// TwinCAT 3 PLC project MC2
// Title: Tc_MC2
// Company: NewEngineer
// Author: Tc_MC2
// ProjectVersion: 0.1.1.1
// Description: https://github.com/phucpha
// ProgramVersion: 3.1.4024.0
// libraries:
//   Tc2_MC2, * (Beckhoff Automation GmbH)
//   Tc2_Standard, * (Beckhoff Automation GmbH)
//   Tc2_System, * (Beckhoff Automation GmbH)
//   Tc3_EventLogger, * (Beckhoff Automation GmbH)
//   Tc3_Mc3Definitions, * (Beckhoff Automation GmbH)
//   Tc3_Module, * (Beckhoff Automation GmbH)
//   Tc_Utilities, * (NewEngineer)
// project tree:
//   DUTs/CAextension/ E_AxisStateCA.TcDUT
//   DUTs/CA/ E_AxesGroupCAMethodState.TcDUT, E_AxesGroupCAState.TcDUT, E_AxesGroupCAStateAborting.TcDUT, E_AxesGroupCAStateInit.TcDUT, E_AxesGroupCAStatePlcOpen.TcDUT
//   DUTs/Universal Axis/ E_AxisJogDirection.TcDUT, E_AxisState.TcDUT, E_AxisStateInit.TcDUT, E_AxisStatePlcOpen.TcDUT
//   DUTs/Visu/ E_VisuCtrlAxisImgType.TcDUT (not stored), E_VisuCtrlAxisJogMode.TcDUT (not stored), E_VisuCtrlSingleAxisState.TcDUT (not stored), ST_VisuCtrlAxisFrame.TcDUT (not stored)
//   POUs/AxesGroup/ FB_AxesGroupCA.TcPOU, I_AxesGroupCA.TcIO
//   POUs/Axis/ FB_AxisServo.TcPOU, FB_AxisServoCA.TcPOU, FB_UniversalAxis.TcPOU, I_UniversalAxis.TcIO, I_UniversalAxisCA.TcIO
//   Version/ Global_Version.TcGVL
// real-time tasks:
//   TASK PlcTask: cycle T#10ms, priority 20, ADS port 350

// ---- DUTs/CAextension/E_AxisStateCA.TcDUT
{attribute 'strict'}
TYPE E_AxisStateCA :
(
	AXIS_CA_IDLE				:= 0,
	AXIS_CA_MOVE_ABSOLUTE 		:= 10,
	AXIS_CA_MOVE_ABSOLUTE_DONE 	:= 20,
	AXIS_CA_MOVE_RELATIVE 		:= 30,
	AXIS_CA_MOVE_RELATIVE_DONE 	:= 40,
	AXIS_CA_HALT				:= 50,
	AXIS_CA_HALT_DONE			:= 60
);
END_TYPE

// ---- DUTs/CA/E_AxesGroupCAMethodState.TcDUT
{attribute 'strict'}
TYPE E_AxesGroupCAMethodState :
(
	AXES_GROUP_METHOD_EXECUTE 	:= 0,	(* Reseting all fubs *)
	AXES_GROUP_METHOD_DONE		:= 10	(* Enabling axes group *)
);
END_TYPE

// ---- DUTs/CA/E_AxesGroupCAState.TcDUT
{attribute 'strict'}
TYPE E_AxesGroupCAState :
(
	AXES_GROUP_UNINITIALIZED 		:= 0,	(* Axes group is disabled, not ready to work *)
	AXES_GROUP_INITIALIZING 		:= 10,	(* Axes group is preprating to work *)
	AXES_GROUP_READY_INITIALIZED	:= 20,	(*  *)
	AXES_GROUP_IDLE 				:= 30,	(* Axes group ready to work, enabled *)
	AXES_GROUP_ADD					:= 40,	(* Adding axis to axes group *)
	AXES_GROUP_ADD_DONE				:= 50,	(* Adding axis to axes group done *)
	AXES_GROUP_REMOVE				:= 60,	(* Removeing axis from axes group *)
	AXES_GROUP_REMOVE_DONE			:= 70,	(* Removing axis from axes group done *)
	AXES_GROUP_REMOVE_ALL			:= 80,	(* Remoing all axis from axes group *)
	AXES_GROUP_REMOVE_ALL_DONE		:= 90,	(* Removing all axis from axes group done *)
	AXES_GROUP_ENABLE				:= 100,	(* Enabling axes group *)
	AXES_GROUP_ENABLE_DONE			:= 110,	(* Enabling axes group done *)
	AXES_GROUP_DISABLE				:= 120,	(* Disabling axes group *)
	AXES_GROUP_DISABLE_DONE			:= 130,	(* Disabling axes group done *)
	AXES_GROUP_RESET				:= 140,	(* Reseting funcion block *)
	AXES_GROUP_RESET_DONE			:= 150,	(* Reseting function block done *)
	AXES_GROUP_HALT					:= 160,	(* Halt axes group *)
	AXES_GROUP_HALT_DONE			:= 170,	(* Halt axes group done *)
	AXES_GROUP_STOP					:= 180,	(* Stop axes group *)
	AXES_GROUP_STOP_DONE			:= 190,	(* Stop axes group done *)
	AXES_GROUP_UNLOCK				:= 200,	(* Unlock axes group after stop *)
	AXES_GROUP_UNLOCK_DONE			:= 210,	(* Unlock axes group after stop done *)
	AXES_GROUP_ABORTING				:= -10	(* Aborting *)
);
END_TYPE

// ---- DUTs/CA/E_AxesGroupCAStateAborting.TcDUT
{attribute 'strict'}
TYPE E_AxesGroupCAStateAborting :
(
	AXES_GROUP_ABORTING_RESET_FBS 		:= 0,	(* Reseting all function blocks used inside function block *)
	AXES_GROUP_ABORTING_REMOVE_ALL		:= 10,	(* Removing all axis from axes group  *)
	AXES_GROUP_ABORTING_RESET_ERRORS	:= 20,	(* Reseting axes group errors *)
	AXES_GROUP_ABORTING_DISABLE			:= 30,	(* Disabling axes group *)
	AXES_GROUP_ABORTING_DONE			:= 40	(* Aborting procedure finished *)
);
END_TYPE

// ---- DUTs/CA/E_AxesGroupCAStateInit.TcDUT
{attribute 'strict'}
TYPE E_AxesGroupCAStateInit :
(
	AXES_GROUP_INIT_RESET 	:= 0,	(* Reseting all fubs *)
	AXES_GROUP_INIT_ENABLE	:= 10,	(* Enabling axes group *)
	AXES_GROUP_INIT_DONE	:= 20	(* Initialization procedure done*)
);
END_TYPE

// ---- DUTs/CA/E_AxesGroupCAStatePlcOpen.TcDUT
{attribute 'strict'}
TYPE E_AxesGroupCAStatePlcOpen :
(
	PLCOPEN_AXES_GROUP_DISABLED 	:= 0,	(* Axes group is disabled *)
	PLCOPEN_AXES_GROUP_NOT_READY 	:= 10,	(* Axes group is not ready to work*)
	PLCOPEN_AXES_GROUP_STANDBY 		:= 20,	(* Axes group is enabled and waiting for commands*)
	PLCOPEN_AXES_GROUP_MOVING 		:= 30,	(* Axes group is moving *)
	PLCOPEN_AXES_GROUP_STOPPING 	:= 40,	(* Axes group is stopping *)
	PLCOPEN_AXES_GROUP_ERROR		:= 50	(* Axes group is in error state*)
);
END_TYPE

// ---- DUTs/Universal Axis/E_AxisJogDirection.TcDUT
{attribute 'strict'}
TYPE E_AxisJogDirection :
(
	AXIS_JOG_DIR_POSITIVE := 0,	(* Perform jog in positive direction *)
	AXIS_JOG_DIR_NEGATIVE := 10	(* Perform jog in negative direction *)
);
END_TYPE

// ---- DUTs/Universal Axis/E_AxisState.TcDUT
{attribute 'strict'}
TYPE E_AxisState :
(
	AXIS_UNINITIALIZED		:= 0,	(* Axis is not prepared to work - power is off *)
	AXIS_INITIALIZING		:= 10,	(* Axis is preparing to power - reset FB and power on *)
	AXIS_READY_INITIALIZED	:= 20,	(*  *)
	AXIS_IDLE				:= 30,	(* Axis is ready for orders *)
	AXIS_HOME				:= 40,	(* Axis is homing to reference point *)
	AXIS_HOME_DONE			:= 50,	(* Axis homing procedure has finished - fererence position has been found *)
	AXIS_MOVE_VELOCITY		:= 60,	(* Axis started continous motion to setpoint velocity - accelerating *)
	AXIS_MOVE_VELOCITY_DONE	:= 70,	(* Axis reached constant setpoint velocity for continous motion *)
	AXIS_MOVE_ABSOLUTE		:= 80,	(* Axis is moving to absolute position - discrete motion *)
	AXIS_MOVE_ABSOLUTE_DONE	:= 90,	(* Axis movement to absolute position finished *)
	AXIS_MOVE_ADDITIVE		:= 100,	(* Axis relative movement by desired distance *)
	AXIS_MOVE_ADDITIVE_DONE	:= 110,	(* Axis relative relative movement by desired distance finished *)
	AXIS_MOVE_RELATIVE		:= 120,	(* Axis relative movement by desired distance *)
	AXIS_MOVE_RELATIVE_DONE	:= 130,	(* Axis relative relative movement by desired distance finished *)
	AXIS_MOVE_JOG			:= 140,	(* Axis manual move using jog function *)
	AXIS_MOVE_JOG_DONE		:= 150,	(* Axis jog done *)
	AXIS_STOP				:= 160,	(* Axis is stopping *)
	AXIS_STOP_DONE			:= 170,	(* Axis stopped *)
	AXIS_HALT				:= 180,	(* Axis halts started motion command *)
	AXIS_HALT_DONE			:= 190,	(* Axis motion halted *)
	AXIS_RESET				:= 200,	(* Axis is resseting all function blocks and occured errors *)
	AXIS_RESET_DONE			:= 210,	(* Axis reset procedure done *)
	AXIS_COUPLE				:= 220, (* Axis is synchronizing to another master axis *)
	AXIS_COUPLE_DONE		:= 230,	(* Axis coupled to another master axis*)
	AXIS_DECOUPLE			:= 240,	(* Axis is decoupling from synchronized motion *)
	AXIS_DECOUPLE_DONE		:= 250,	(* Axis decoupled from synchronizing motion*)
	AXIS_UNLOCK				:= 260,	(* Axis is unlocking after stop command *)
	AXIS_UNLOCK_DONE		:= 270,	(* Axis unlocked after stop command *)
	AXIS_EXTENSION			:= 999,	(* Special state used by child FB's to implement additional states *)
	AXIS_ABORTING			:= -10	(* Aborting *)
);
END_TYPE

// ---- DUTs/Universal Axis/E_AxisStateInit.TcDUT
{attribute 'strict'}
TYPE E_AxisStateInit :
(
	AXIS_INIT_RESET		:= 0,	(* Reseting all function blocks *)
	AXIS_INIT_POWER_ON	:= 10,	(* Powering on the axis *)
	AXIS_INIT_DONE		:= 20	(* Initialization done *)
);
END_TYPE

// ---- DUTs/Universal Axis/E_AxisStatePlcOpen.TcDUT
{attribute 'strict'}
TYPE E_AxisStatePlcOpen :
(
	AXIS_PLCOPEN_DISABLED				:= 0,	(* Axis power controler if of *)
	AXIS_PLCOPEN_STANDSTILL				:= 10,	(* Axis is powered on *)
	AXIS_PLCOPEN_HOMING					:= 20,	(* Axis performs homing procedure *)
	AXIS_PLCOPEN_STOPPING				:= 30,	(* Axis is stopping the movement *)
	AXIS_PLCOPEN_CONTINUOUS_MOTION		:= 40,	(* Axis is moving continuosly with constant speed *)
	AXIS_PLCOPEN_DISCRETE_MOTION		:= 50,	(* Axis is moving from point to point *)
	AXIS_PLCOPEN_SYNCHRONIZED_MOTION 	:= 60,	(* Axis is moving in synchronized motion to master *)
	AXIS_PLCOPEN_ERRORSTOP				:= 70	(* Axis stoped because of error *)
);
END_TYPE

// ---- Version/Global_Version.TcGVL
{attribute 'TcGenerated'}
{attribute 'no-analysis'}
{attribute 'linkalways'}
// This function has been automatically generated from the project information.
VAR_GLOBAL CONSTANT
	{attribute 'const_non_replaced'}
	stLibVersion_Tc_MC2 : ST_LibVersion := (iMajor := 0, iMinor := 1, iBuild := 1, iRevision := 1, nFlags := 0, sVersion := '0.1.1.1');
END_VAR

// ---- POUs/AxesGroup/I_AxesGroupCA.TcIO
INTERFACE I_AxesGroupCA

PROPERTY Active : REFERENCE TO BOOL
GET
END_GET
END_PROPERTY

PROPERTY AxesGroupRef : REFERENCE TO AXES_GROUP_REF
GET
END_GET
END_PROPERTY

PROPERTY AxesInGroup : REFERENCE TO UINT
GET
END_GET
END_PROPERTY

PROPERTY AxisAdded : REFERENCE TO BOOL
GET
END_GET
END_PROPERTY

PROPERTY AxisRemoved : REFERENCE TO BOOL
GET
END_GET
END_PROPERTY

PROPERTY Busy : REFERENCE TO BOOL
GET
END_GET
END_PROPERTY

PROPERTY Deceleration : LREAL
GET
END_GET
SET
END_SET
END_PROPERTY

PROPERTY Error : REFERENCE TO BOOL
GET
END_GET
END_PROPERTY

PROPERTY ErrorID : REFERENCE TO UDINT
GET
END_GET
END_PROPERTY

PROPERTY GroupEnabled : REFERENCE TO BOOL
GET
END_GET
END_PROPERTY

PROPERTY GroupLocked : REFERENCE TO BOOL
GET
END_GET
END_PROPERTY

PROPERTY Jerk : LREAL
GET
END_GET
SET
END_SET
END_PROPERTY

METHOD MR_Abort : BOOL
VAR_INPUT
END_VAR
END_METHOD

METHOD MR_Add : BOOL
VAR_INPUT
	stInternalAxisRef	: AXIS_REF;
	iAxisIdentyficator	: UINT;
END_VAR
END_METHOD

METHOD MR_Disable : BOOL
VAR_INPUT
END_VAR
END_METHOD

METHOD MR_Enable : BOOL
VAR_INPUT
END_VAR
END_METHOD

METHOD MR_FirstCycle
VAR_INPUT
	sName 			: STRING;	(* Default axes group object name *)
	lrDeceleration 	: LREAL;	(* Default axes group object deceleration *)
	lrJerk			: LREAL;	(* Default axes group object jerk *)
END_VAR
END_METHOD

METHOD MR_Halt : BOOL
VAR_INPUT
END_VAR
END_METHOD

METHOD MR_Init : BOOL
VAR_INPUT
END_VAR
END_METHOD

METHOD MR_Remove : BOOL
VAR_INPUT
	iAxisIdentyficator	: UINT;
END_VAR
END_METHOD

METHOD MR_RemoveAll : BOOL
VAR_INPUT
END_VAR
END_METHOD

METHOD MR_Reset : BOOL
VAR_INPUT
END_VAR
END_METHOD

METHOD MR_Stop : BOOL
VAR_INPUT
END_VAR
END_METHOD

METHOD MR_Unlock : BOOL
VAR_INPUT
END_VAR
END_METHOD

PROPERTY Name : STRING
GET
END_GET
SET
END_SET
END_PROPERTY

PROPERTY RemovedAll : REFERENCE TO BOOL
GET
END_GET
END_PROPERTY

PROPERTY State : REFERENCE TO E_AxesGroupCAState
GET
END_GET
END_PROPERTY

PROPERTY StatePlcOpen : REFERENCE TO E_AxesGroupCAStatePlcOpen
GET
END_GET
END_PROPERTY

END_INTERFACE

// ---- POUs/Axis/I_UniversalAxis.TcIO
INTERFACE I_UniversalAxis

PROPERTY Acceleration : LREAL
GET
END_GET
SET
END_SET
END_PROPERTY

PROPERTY Active : REFERENCE TO BOOL
GET
END_GET
END_PROPERTY

PROPERTY ActualPosition : REFERENCE TO LREAL
GET
END_GET
END_PROPERTY

PROPERTY ActualVelocity : REFERENCE TO LREAL
GET
END_GET
END_PROPERTY

PROPERTY AxisErrorID : REFERENCE TO UDINT
GET
END_GET
END_PROPERTY

PROPERTY AxisRef : AXIS_REF
GET
END_GET
SET
END_SET
END_PROPERTY

PROPERTY BufferMode : MC_BufferMode
GET
END_GET
SET
END_SET
END_PROPERTY

PROPERTY Busy : REFERENCE TO BOOL
GET
END_GET
END_PROPERTY

PROPERTY Deceleration : LREAL
GET
END_GET
SET
END_SET
END_PROPERTY

PROPERTY Direction : Tc2_MC2.MC_Direction
GET
END_GET
SET
END_SET
END_PROPERTY

PROPERTY Error : REFERENCE TO BOOL
GET
END_GET
END_PROPERTY

PROPERTY ErrorID : REFERENCE TO UDINT
GET
END_GET
END_PROPERTY

PROPERTY Halted : REFERENCE TO BOOL
GET
END_GET
END_PROPERTY

PROPERTY InPosition : REFERENCE TO BOOL
GET
END_GET
END_PROPERTY

PROPERTY InVelocity : REFERENCE TO BOOL
GET
END_GET
END_PROPERTY

PROPERTY IsHomed : REFERENCE TO BOOL
GET
END_GET
END_PROPERTY

PROPERTY Jerk : LREAL
GET
END_GET
SET
END_SET
END_PROPERTY

PROPERTY JogAcceleration : LREAL
GET
END_GET
SET
END_SET
END_PROPERTY

PROPERTY JogDeceleration : LREAL
GET
END_GET
SET
END_SET
END_PROPERTY

PROPERTY JogDirection : E_AxisJogDirection
GET
END_GET
SET
END_SET
END_PROPERTY

PROPERTY JogDone : REFERENCE TO BOOL
GET
END_GET
END_PROPERTY

PROPERTY JogJerk : LREAL
GET
END_GET
SET
END_SET
END_PROPERTY

PROPERTY JogMode : E_JogMode
GET
END_GET
SET
END_SET
END_PROPERTY

PROPERTY JogPosition : LREAL
GET
END_GET
SET
END_SET
END_PROPERTY

PROPERTY JogVelocity : LREAL
GET
END_GET
SET
END_SET
END_PROPERTY

PROPERTY LagError : LREAL
GET
END_GET
END_PROPERTY

PROPERTY MoveActive : REFERENCE TO BOOL
GET
END_GET
END_PROPERTY

METHOD MR_Abort : BOOL
END_METHOD

METHOD MR_FirstCycle
VAR_INPUT
	sName 				: STRING; 	(* Axis object name *)
	sMeasurementUnits	: STRING;	(* Measurement units used by axis *)
	bModulo				: BOOL;		(* Axis is periodic *)
END_VAR
END_METHOD

METHOD MR_Halt : BOOL
END_METHOD

METHOD MR_Home : BOOL
VAR_INPUT
	lrHomePosition : LREAL;
END_VAR
END_METHOD

METHOD MR_Init : BOOL
END_METHOD

METHOD MR_Jog : BOOL
VAR_INPUT
	//lrJogPosition : LREAL;
	//eJogDirection : E_AxisJogDirection;
	//eJogMode	  : E_JogMode;
	bJogActive	  : BOOL;
END_VAR
END_METHOD

METHOD MR_MoveAbsolute : BOOL
VAR_INPUT
	lrAbsolutePosition : LREAL;
END_VAR
END_METHOD

METHOD MR_MoveAdditive : BOOL
VAR_INPUT
	lrRelativeDistance : LREAL;
END_VAR
END_METHOD

METHOD MR_MoveRelative : BOOL
VAR_INPUT
	lrRelativeDistance : LREAL;
END_VAR
END_METHOD

METHOD MR_MoveVelocity : BOOL
END_METHOD

METHOD MR_Reset : BOOL
END_METHOD

METHOD MR_Stop : BOOL
END_METHOD

PROPERTY Name : STRING
GET
END_GET
SET
END_SET
END_PROPERTY

PROPERTY Options : ST_MoveOptions
GET
END_GET
SET
END_SET
END_PROPERTY

PROPERTY Override : LREAL
GET
END_GET
SET
END_SET
END_PROPERTY

PROPERTY PowerOn : REFERENCE TO BOOL
GET
END_GET
END_PROPERTY

PROPERTY SetpointPosition : LREAL
GET
END_GET
END_PROPERTY

PROPERTY SetpointVelocity : LREAL
GET
END_GET
END_PROPERTY

PROPERTY State : REFERENCE TO E_AxisState
GET
END_GET
END_PROPERTY

PROPERTY StatePlcOpen : REFERENCE TO E_AxisStatePlcOpen
GET
END_GET
END_PROPERTY

PROPERTY StopDeceleration : LREAL
GET
END_GET
SET
END_SET
END_PROPERTY

PROPERTY StopJerk : LREAL
GET
END_GET
SET
END_SET
END_PROPERTY

PROPERTY Stopped : REFERENCE TO BOOL
GET
END_GET
END_PROPERTY

PROPERTY Unit : STRING
GET
END_GET
SET
END_SET
END_PROPERTY

PROPERTY Velocity : LREAL
GET
END_GET
SET
END_SET
END_PROPERTY

END_INTERFACE

// ---- POUs/Axis/I_UniversalAxisCA.TcIO
INTERFACE I_UniversalAxisCA EXTENDS I_UniversalAxis

PROPERTY DirectionCA : Tc3_Mc3Definitions.MC_DIRECTION
GET
END_GET
SET
END_SET
END_PROPERTY

PROPERTY Gap : MC_LREAL
GET
END_GET
SET
END_SET
END_PROPERTY

PROPERTY HaltedCA : REFERENCE TO BOOL
GET
END_GET
END_PROPERTY

METHOD MR_HaltCA : BOOL
VAR_INPUT
END_VAR
END_METHOD

METHOD MR_MoveAbsoluteCA : BOOL
VAR_INPUT
	lrAbsolutePosition : LREAL;
END_VAR
END_METHOD

METHOD MR_MoveRelativeCA : BOOL
VAR_INPUT
	lrRelativeDistance : LREAL;
END_VAR
END_METHOD

PROPERTY StateCA : REFERENCE TO E_AxisStateCA
GET
END_GET
END_PROPERTY

END_INTERFACE

// ---- POUs/AxesGroup/FB_AxesGroupCA.TcPOU
(*
:Description: This function block is used to control collision avoidance axes group.
*)
FUNCTION_BLOCK FB_AxesGroupCA IMPLEMENTS I_AxesGroupCA
VAR
	bFirstCycle				: BOOL := TRUE;						(* First cycle bit *)	
	sName 					: STRING;							(* Axes group name for other utilities *)
	
	(* Hardware links *)
	stAxesGroupRef 			: AXES_GROUP_REF;					(* Axes group reference object *)
	stInternalAxisRef 		: AXIS_REF;							(* Internal axis reference object *)
	
	(* Internal commands *)
	bInit 					: BOOL;								(* Power on axis and prepare to work *)
	bAbort 					: BOOL;								(* Power off axis and reset status flags *)
	bReset 					: BOOL;								(* Reset axis and return to READY state *)
	bAdd 					: BOOL;								(* Add axis to the group *)
	bRemove 				: BOOL;								(* Remove axis from the group *)
	bRemoveAll 				: BOOL;								(* Remove all axes from the group *)
	bEnable 				: BOOL;								(* Enable the group *)
	bDisable 				: BOOL;								(* Disable the group *)
	bGroupHalt				: BOOL;								(* Halt all axes in group *)
	bGroupStop				: BOOL;								(* Stop all axes in group *)
	bGroupUnlock			: BOOL;								(* Unlock axes group after stop *)
	
	(* Internal parameters *)
	iIdentInGroup			: UDINT;							(* An axis identyficator *)
	lrDeceleration			: LREAL;							(* Decelearion of all axes in group *)
	lrJerk					: LREAL;							(* Jerk of all axes in group *)
	
	(* Internal status *)
	bActive					: BOOL;
	bBusy					: BOOL;								(* Function block currently executes one of the requests *)
	bError 					: BOOL;								(* Error status flag *)
	iErrorID 				: UDINT;							(* Error ID *)
	bResetDone				: BOOL;								(* All internal errors of a group and all axes belonging to the group reset *)	
	bAxisAdded				: BOOL;								(* Axis added to the group *)
	bAxisRemoved			: BOOL;								(* Axis removed from the group *)
	bRemovedAll				: BOOL;								(* Removing all axes and disabling the group *)
	bGroupEnabled			: BOOL;								(* Axes group enabled *)
	bGroupHalted			: BOOL;								(* Axes group halted *)
	bGroupStopped			: BOOL;								(* Axes group stopped *)
	iAxesInGroup			: UINT;								(* Amount of the axes in the group *)
	bGroupLocked			: BOOL;								(* Group locked by stop function *)
	eStatePlcOpen 			: E_AxesGroupCAStatePlcOpen;
	eAxesGroupState 		: E_AxesGroupCAState;
	eAxesGroupStateInit		: E_AxesGroupCAStateInit;
	eAxesGroupStateAbort	: E_AxesGroupCAStateAborting;
	eAxesGroupMethodState	: E_AxesGroupCAMethodState;
	
	
	(* Function blocks *)
	fbMcAddAxisToGroup		: MC_AddAxisToGroup;				(* FB to add an axis to the group *)
	fbMcRemoveAxisFromGroup	: MC_RemoveAxisFromGroup;			(* FB to remove an axis from the group *)
	fbMcUngroupAllAxes 		: MC_UngroupAllAxes;				(* FB to ungroup all axes from the group *)
	
	fbMcGroupEnable 		: MC_GroupEnable;					(* FB to enable the group *)
	fbMcGroupDisable 		: MC_GroupDisable;					(* FB to disable the group *)
	
	fbMcGroupReadStatus		: MC_GroupReadStatus;				(* FB to read current axes group status *)
	fbMcGroupReadError		: MC_GroupReadError;				(* FB to read axes group error *)
	fbMcGroupReset 			: MC_GroupReset;					(* FB to reset axes group *)
	
	fbMcGroupHalt			: MC_GroupHalt;						(* FB to halt all axes in group *)
	fbMcGroupStop			: MC_GroupStop;						(* FB to stop all axes in group *)
	
	(* Tc3 EventLogger - messages *)
	fbAlarmGroupReset		: FB_TcAlarm;						(*  *)
	fbAlarmUngroupAll		: FB_TcAlarm;						(*  *)
	fbAlarmGroupDisable		: FB_TcAlarm;						(*  *)
	fbAlarmAddAxisToGroup	: FB_TcAlarm;						(*  *)
	fbAlarmGroupEnable		: FB_TcAlarm;						(*  *)
	fbAlarmRemoveFromGroup	: FB_TcAlarm;						(*  *)
	
	bResetConfirmation 		: BOOL;
	bGroupHaltLog			: BOOL;
	bGroupStopLog			: BOOL;
	
	rtError					: R_TRIG; 				(* Rising edge trigger for function block error *)
	
END_VAR

(* Run first cycle procedure *)
IF bFirstCycle THEN
	bFirstCycle := FALSE;
		
	fbAlarmGroupReset.CreateEx( stEventEntry := TC_EVENTS.ShellAxesGroupEventClass.GroupReset, 
									bWithConfirmation := 1,
									ipSourceInfo := 0);
									
	fbAlarmUngroupAll.CreateEx( stEventEntry := TC_EVENTS.ShellAxesGroupEventClass.UngroupAll, 
									bWithConfirmation := 1,
									ipSourceInfo := 0);
		
	fbAlarmGroupDisable.CreateEx( stEventEntry := TC_EVENTS.ShellAxesGroupEventClass.GroupDisable, 
									bWithConfirmation := 1,
									ipSourceInfo := 0);
									
	fbAlarmAddAxisToGroup.CreateEx( stEventEntry := TC_EVENTS.ShellAxesGroupEventClass.AddAxisToGroup, 
									bWithConfirmation := 1,
									ipSourceInfo := 0);
		
	fbAlarmGroupEnable.CreateEx( stEventEntry := TC_EVENTS.ShellAxesGroupEventClass.GroupEnable, 
									bWithConfirmation := 1,
									ipSourceInfo := 0);
									
	fbAlarmRemoveFromGroup.CreateEx( stEventEntry := TC_EVENTS.ShellAxesGroupEventClass.RemoveFromGroup, 
									bWithConfirmation := 1,
									ipSourceInfo := 0);
									
END_IF

(* Reading the group status from group reference *)
fbMcGroupReadStatus( AxesGroup := stAxesGroupRef, Enable := TRUE);

(* Setting the PLCOpen group status*)
IF fbMcGroupReadStatus.Valid THEN
	IF fbMcGroupReadStatus.GroupDisabled THEN
		eStatePlcOpen := PLCOPEN_AXES_GROUP_DISABLED;
		
	ELSIF fbMcGroupReadStatus.GroupErrorStop THEN
		eStatePlcOpen := PLCOPEN_AXES_GROUP_ERROR;
		
	ELSIF fbMcGroupReadStatus.GroupStandby THEN
		eStatePlcOpen := PLCOPEN_AXES_GROUP_STANDBY;
		
	ELSIF fbMcGroupReadStatus.GroupMoving THEN
		eStatePlcOpen := PLCOPEN_AXES_GROUP_MOVING;
		
	ELSIF fbMcGroupReadStatus.GroupStopping THEN
		eStatePlcOpen := PLCOPEN_AXES_GROUP_STOPPING;
		
	END_IF
END_IF

(* Reading errors *)
fbMcGroupReadError( AxesGroup := stAxesGroupRef, Enable := TRUE);

IF fbMcGroupReadError.Valid THEN
	iErrorID := fbMcGroupReadError.GroupErrorId;
END_IF


(* Report errors that occur *)
rtError(CLK:=bError);

IF rtError.Q THEN 
	fbMachineLogger.MR_AddLogs(FUN_MergeStrings5(sName, ' : Error occured (error ID: ', UDINT_TO_STRING(iErrorID), ')', ''));

END_IF

(* Execute state machine *)
StateMachine();

PROPERTY Active : REFERENCE TO BOOL
GET
Active REF= bActive;
END_GET
END_PROPERTY

PROPERTY AxesGroupRef : REFERENCE TO Tc3_McCoordinatedMotion.AXES_GROUP_REF
GET
AxesGroupRef REF= stAxesGroupRef;
END_GET
END_PROPERTY

PROPERTY AxesInGroup : REFERENCE TO UINT
GET
AxesInGroup REF= iAxesInGroup;
END_GET
END_PROPERTY

PROPERTY AxisAdded : REFERENCE TO BOOL
GET
AxisAdded REF= bAxisAdded;
END_GET
END_PROPERTY

PROPERTY AxisRemoved : REFERENCE TO BOOL
GET
AxisRemoved REF= bAxisRemoved;
END_GET
END_PROPERTY

PROPERTY Busy : REFERENCE TO BOOL
GET
Busy REF= bBusy;
END_GET
END_PROPERTY

(* Decelearion of all axes in group *)
PROPERTY Deceleration : LREAL
GET
Deceleration := lrDeceleration;
END_GET
SET
lrDeceleration := Deceleration;
END_SET
END_PROPERTY

PROPERTY Error : REFERENCE TO BOOL
GET
Error REF= bError;
END_GET
END_PROPERTY

PROPERTY ErrorID : REFERENCE TO UDINT
GET
ErrorID REF= iErrorID;
END_GET
END_PROPERTY

PROPERTY GroupEnabled : REFERENCE TO BOOL
GET
GroupEnabled REF= bGroupEnabled;
END_GET
END_PROPERTY

PROPERTY GroupHalted : REFERENCE TO BOOL
GET
GroupHalted REF= bGroupHalted;
END_GET
END_PROPERTY

PROPERTY GroupLocked : REFERENCE TO BOOL
GET
GroupLocked REF= bGroupLocked;
END_GET
END_PROPERTY

PROPERTY GroupStopped : REFERENCE TO BOOL
GET
GroupStopped REF= bGroupStopped;
END_GET
END_PROPERTY

(* Jerk of all axes in group *)
PROPERTY Jerk : LREAL
GET
Jerk := lrJerk;
END_GET
SET
lrJerk := Jerk;
END_SET
END_PROPERTY

METHOD MR_Abort : BOOL
IF eAxesGroupState >= AXES_GROUP_IDLE THEN
	bBusy := TRUE;
	bAbort := TRUE;
	eAxesGroupStateAbort := AXES_GROUP_ABORTING_RESET_FBS;
	eAxesGroupState := AXES_GROUP_ABORTING;	
	
	fbMachineLogger.MR_AddLogs(CONCAT(sName,' : abort requested'));			

ELSIF eAxesGroupState = AXES_GROUP_ABORTING AND eAxesGroupStateAbort = AXES_GROUP_ABORTING_DONE THEN
	bActive := FALSE;
	bAbort := FALSE;	
	MR_Abort := TRUE;
	bBusy := FALSE;
	
	fbMachineLogger.MR_AddLogs(CONCAT(sName,' : abort done'));	

END_IF
END_METHOD

METHOD MR_Add : BOOL
VAR_INPUT
	stInternalAxisRef	: AXIS_REF;
	iAxisIdentyficator	: UINT;
END_VAR
IF eAxesGroupState = AXES_GROUP_IDLE THEN
	bBusy 			:= TRUE;
	bAdd 			:= TRUE;
	
	bAxisAdded 		:= FALSE;
	bAxisRemoved 	:= FALSE;
	bRemovedAll 	:= FALSE;
	bResetDone		:= FALSE;
	
	THIS^.stInternalAxisRef := stInternalAxisRef;
	iIdentInGroup := iAxisIdentyficator;
	
	eAxesGroupState := AXES_GROUP_ADD;
	fbMachineLogger.MR_AddLogs(CONCAT(sName,' : axes group addition requested'));			
	
ELSIF eAxesGroupState = AXES_GROUP_ADD_DONE THEN
	bAdd 			:= FALSE;
	
	MR_Add 			:= TRUE;
	bAxisAdded 		:= TRUE;
	iAxesInGroup 	:= iAxesInGroup + 1;

	bBusy			:= FALSE;

	fbMachineLogger.MR_AddLogs(CONCAT(sName,' : axes group addition done'));			
	
END_IF
END_METHOD

METHOD MR_Disable : BOOL
VAR_INPUT
END_VAR
IF eAxesGroupState = AXES_GROUP_IDLE THEN
	bBusy 			:= TRUE;
	bDisable 		:= TRUE;
	
	bAxisAdded 		:= FALSE;
	bAxisRemoved 	:= FALSE;
	bRemovedAll 	:= FALSE;
	bResetDone		:= FALSE;
	
	eAxesGroupState := AXES_GROUP_DISABLE;
	fbMachineLogger.MR_AddLogs(CONCAT(sName,' : axes group disablement requested'));				
	
ELSIF eAxesGroupState = AXES_GROUP_DISABLE_DONE THEN
	bDisable 		:= FALSE;
	
	MR_Disable 		:= TRUE;
	bGroupEnabled	:= FALSE;
	
	bBusy 			:= FALSE;
	
	fbMachineLogger.MR_AddLogs(CONCAT(sName,' : axes group disablement done'));			
	
END_IF
END_METHOD

METHOD MR_Enable : BOOL
VAR_INPUT
END_VAR
IF eAxesGroupState = AXES_GROUP_IDLE THEN
	bBusy			:= TRUE;
	bEnable 		:= TRUE;
	
	bAxisAdded 		:= FALSE;
	bAxisRemoved 	:= FALSE;
	bRemovedAll 	:= FALSE;
	bResetDone		:= FALSE;
	
	eAxesGroupState := AXES_GROUP_ENABLE;
	fbMachineLogger.MR_AddLogs(CONCAT(sName,' : axes group enablement requested'));
	
ELSIF eAxesGroupState = AXES_GROUP_ENABLE_DONE THEN
	bEnable 		:= FALSE;
	MR_Enable 		:= TRUE;
	bGroupEnabled 	:= TRUE;
	bBusy 			:= FALSE;
	fbMachineLogger.MR_AddLogs(CONCAT(sName,' : axes group enablement done'));
	
END_IF
END_METHOD

METHOD MR_FirstCycle
VAR_INPUT
	sName 			: STRING;	(* Default axes group object name *)
	lrDeceleration 	: LREAL;	(* Default axes group object deceleration *)
	lrJerk			: LREAL;	(* Default axes group object jerk *)
END_VAR
THIS^.sName := sName;
THIS^.lrDeceleration := lrDeceleration;
THIS^.lrJerk := lrJerk;
END_METHOD

METHOD MR_Halt : BOOL
VAR_INPUT
END_VAR
IF eAxesGroupState >= AXES_GROUP_IDLE AND eAxesGroupState <> AXES_GROUP_HALT_DONE THEN
	bBusy := TRUE;
	
	IF NOT bGroupHaltLog THEN 
		fbMachineLogger.MR_AddLogs(CONCAT(sName,' : halt requested'));
		bGroupHaltLog := TRUE;
	END_IF
	
	bGroupHalt := TRUE;
	MR_Halt := FALSE;
	eAxesGroupState := AXES_GROUP_HALT;
	
ELSIF eAxesGroupState = AXES_GROUP_HALT_DONE THEN
	bGroupHalt := FALSE;
	MR_Halt := TRUE;
	bGroupHaltLog := FALSE;
	bBusy := FALSE;
	
	fbMachineLogger.MR_AddLogs(CONCAT(sName,' : halt done'));
	
END_IF
END_METHOD

METHOD MR_Init : BOOL
IF eAxesGroupState = AXES_GROUP_UNINITIALIZED THEN
	bBusy := TRUE;
	bActive := TRUE;
	bInit := TRUE;
	MR_Init := FALSE;
	eAxesGroupState := AXES_GROUP_INITIALIZING;
	fbMachineLogger.MR_AddLogs(CONCAT(sName,' : initialization requested'));
	
ELSIF eAxesGroupState = AXES_GROUP_INITIALIZING AND eAxesGroupStateInit = AXES_GROUP_INIT_DONE THEN
	bInit := FALSE;
	MR_Init := TRUE;
	bBusy := FALSE;

	fbMachineLogger.MR_AddLogs(CONCAT(sName,' : initialization done'));	

END_IF
END_METHOD

METHOD MR_Remove : BOOL
VAR_INPUT
	iAxisIdentyficator	: UINT;
END_VAR
IF eAxesGroupState = AXES_GROUP_IDLE THEN
	bBusy 			:= TRUE;	
	bRemove 		:= TRUE;
	
	bAxisAdded 		:= FALSE;
	bAxisRemoved 	:= FALSE;
	bRemovedAll 	:= FALSE;
	bResetDone		:= FALSE;
	
	iIdentInGroup	:= iAxisIdentyficator;
	
	eAxesGroupState := AXES_GROUP_REMOVE;
	fbMachineLogger.MR_AddLogs(CONCAT(sName,' : axes group removal requested'));
	
ELSIF eAxesGroupState = AXES_GROUP_REMOVE_DONE THEN
	bRemove 		:= FALSE;
	MR_Remove 		:= TRUE;	
	bAxisRemoved 	:= TRUE;
	iAxesInGroup 	:= iAxesInGroup - 1;
	bBusy 			:= FALSE;
	fbMachineLogger.MR_AddLogs(CONCAT(sName,' : axes group removal done'));
	
END_IF
END_METHOD

METHOD MR_RemoveAll : BOOL
IF eAxesGroupState = AXES_GROUP_IDLE THEN
	bBusy := TRUE;
	bRemoveAll 		:= TRUE;
	
	bAxisAdded 		:= FALSE;
	bAxisRemoved 	:= FALSE;
	bRemovedAll 	:= FALSE;
	bResetDone		:= FALSE;
	
	eAxesGroupState := AXES_GROUP_REMOVE_ALL;
	fbMachineLogger.MR_AddLogs(CONCAT(sName,' : all axes groups removal requested'));
	
ELSIF eAxesGroupState = AXES_GROUP_REMOVE_ALL_DONE THEN
	bRemoveAll 		:= FALSE;
	MR_RemoveAll 	:= TRUE;
	bRemovedAll 	:= TRUE;
	iAxesInGroup 	:= 0;
	bBusy 			:= FALSE;
	
	fbMachineLogger.MR_AddLogs(CONCAT(sName,' : all axes groups removal done'));
	
END_IF
END_METHOD

METHOD MR_Reset : BOOL
IF eAxesGroupState >= AXES_GROUP_IDLE AND eAxesGroupState <> AXES_GROUP_RESET_DONE AND bError THEN
	bBusy			:= TRUE;
	bReset 			:= TRUE;
	bAxisAdded 		:= FALSE;
	bAxisRemoved 	:= FALSE;
	bRemovedAll 	:= FALSE;
	bGroupEnabled 	:= FALSE;
	bResetDone		:= FALSE;
	
	eAxesGroupState := AXES_GROUP_RESET;
	fbMachineLogger.MR_AddLogs(CONCAT(sName,' : reset requested'));
	
ELSIF eAxesGroupState = AXES_GROUP_RESET_DONE THEN
	bReset 		:= FALSE;
	MR_Reset 	:= FALSE;
	bResetDone 	:= TRUE;
	bBusy		:= FALSE;
	
	fbMachineLogger.MR_AddLogs(CONCAT(sName,' : reset done'));
	
END_IF
END_METHOD

METHOD MR_Stop : BOOL
VAR_INPUT
END_VAR
IF eAxesGroupState >= AXES_GROUP_IDLE AND eAxesGroupState <> AXES_GROUP_STOP_DONE THEN
	bBusy := TRUE;
	
	IF NOT bGroupStopLog THEN 
		fbMachineLogger.MR_AddLogs(CONCAT(sName,' : stop requested'));
		bGroupStopLog := TRUE;
	END_IF
	
	bGroupStop := TRUE;
	MR_Stop := FALSE;
	eAxesGroupState := AXES_GROUP_STOP;
	
ELSIF eAxesGroupState = AXES_GROUP_STOP_DONE THEN
	bGroupStop := FALSE;
	MR_Stop := TRUE;
	bGroupLocked := TRUE;
	bGroupStopLog := FALSE;
	bBusy := FALSE;
	fbMachineLogger.MR_AddLogs(CONCAT(sName,' : stop done'));
	
END_IF
END_METHOD

METHOD MR_Unlock : BOOL
VAR_INPUT
END_VAR
IF eAxesGroupState = AXES_GROUP_IDLE AND bGroupLocked THEN
	bBusy := TRUE;
	bGroupUnlock := TRUE;
	MR_Unlock := FALSE;
	eAxesGroupState := AXES_GROUP_UNLOCK;
	
ELSIF eAxesGroupState = AXES_GROUP_UNLOCK_DONE THEN
	bGroupUnlock := FALSE;
	MR_Unlock := TRUE;
	bGroupLocked := FALSE;
	bBusy := FALSE;
	
END_IF
END_METHOD

METHOD PROTECTED MS_Aborting
CASE eAxesGroupStateAbort OF
	AXES_GROUP_ABORTING_RESET_FBS:
		fbMcAddAxisToGroup( AxesGroup := stAxesGroupRef, Axis := stInternalAxisRef, Execute := FALSE);

		fbMcRemoveAxisFromGroup( AxesGroup := stAxesGroupRef, Execute := FALSE);

		fbMcUngroupAllAxes( AxesGroup := stAxesGroupRef, Execute := FALSE);

		fbMcGroupEnable( AxesGroup := stAxesGroupRef, Execute := FALSE);

		fbMcGroupDisable( AxesGroup := stAxesGroupRef, Execute := FALSE);

		fbMcGroupReadStatus( AxesGroup := stAxesGroupRef, Enable := FALSE);

		fbMcGroupReadError( AxesGroup := stAxesGroupRef, Enable := FALSE);
		
		fbMcGroupReset( AxesGroup := stAxesGroupRef, Execute := FALSE);
		
		fbMcGroupHalt( AxesGroup := stAxesGroupRef, Execute := FALSE);
		
		fbMcGroupStop( AxesGroup := stAxesGroupRef, Execute := FALSE);
		
		IF NOT fbMcGroupStop.Busy THEN
			eAxesGroupStateAbort := AXES_GROUP_ABORTING_RESET_ERRORS;
		END_IF
		
	AXES_GROUP_ABORTING_RESET_ERRORS:
		fbMcGroupReset( AxesGroup := stAxesGroupRef, Execute := TRUE);
	
		IF fbMcGroupReset.Error THEN
			bError := TRUE;
			iErrorID := fbMcGroupReset.ErrorID;
			fbMcGroupReset(AxesGroup := stAxesGroupRef, Execute := FALSE);
			
			fbAlarmGroupReset.ipArguments.Clear().AddUDInt(iErrorID);
			fbAlarmGroupReset.Raise(0);
			
		ELSIF fbMcGroupReset.Done THEN
			fbMcGroupReset(AxesGroup := stAxesGroupRef, Execute := FALSE);
			eAxesGroupStateAbort := AXES_GROUP_ABORTING_REMOVE_ALL;
		END_IF
	
	AXES_GROUP_ABORTING_REMOVE_ALL:
		fbMcUngroupAllAxes( AxesGroup := stAxesGroupRef, Execute := TRUE);

		IF fbMcUngroupAllAxes.Error THEN
			bError := TRUE;
			iErrorID := fbMcUngroupAllAxes.ErrorID;
			fbMcUngroupAllAxes( AxesGroup := stAxesGroupRef, Execute := FALSE);
			
			fbAlarmUngroupAll.ipArguments.Clear().AddUDInt(iErrorID);
			fbAlarmUngroupAll.Raise(0);
			
		ELSIF fbMcUngroupAllAxes.Done THEN
			fbMcUngroupAllAxes( AxesGroup := stAxesGroupRef, Execute := FALSE);
			eAxesGroupStateAbort := AXES_GROUP_ABORTING_DISABLE;
		END_IF
	
	AXES_GROUP_ABORTING_DISABLE:
		
		fbMcGroupDisable( AxesGroup := stAxesGroupRef, Execute := TRUE);
	
		IF fbMcGroupDisable.Error THEN
			bError := TRUE;
			iErrorID := fbMcGroupDisable.ErrorID;
			fbMcGroupDisable( AxesGroup := stAxesGroupRef, Execute := FALSE);
			
			fbAlarmGroupDisable.ipArguments.Clear().AddUDInt(iErrorID);
			fbAlarmGroupDisable.Raise(0);
			
		ELSIF fbMcGroupDisable.Done THEN
			fbMcGroupDisable( AxesGroup := stAxesGroupRef, Execute := FALSE);
			eAxesGroupStateAbort := AXES_GROUP_ABORTING_DONE;
		END_IF
	
	AXES_GROUP_ABORTING_DONE:
		IF NOT bAbort THEN
			eAxesGroupState := AXES_GROUP_UNINITIALIZED;
		END_IF
END_CASE
END_METHOD

METHOD PROTECTED MS_Add
CASE eAxesGroupMethodState OF
	AXES_GROUP_METHOD_EXECUTE:
		fbMcAddAxisToGroup( AxesGroup 		:= stAxesGroupRef,
							Axis 			:= stInternalAxisRef,
							Execute 		:= TRUE,
							IdentInGroup 	:= UDINT_TO_IDENTINGROUP(iIdentInGroup));
	
		IF NOT fbMcAddAxisToGroup.Busy THEN
			eAxesGroupMethodState := AXES_GROUP_METHOD_DONE; 
			
		END_IF
	
	AXES_GROUP_METHOD_DONE:
	IF fbMcAddAxisToGroup.Error THEN
		bError := TRUE;
		iErrorID := fbMcAddAxisToGroup.ErrorID;
		fbMcAddAxisToGroup( AxesGroup 		:= stAxesGroupRef,
							Axis 			:= stInternalAxisRef,
							Execute 		:= FALSE);
		
		fbAlarmAddAxisToGroup.ipArguments.Clear().AddUDInt(iErrorID);
		fbAlarmAddAxisToGroup.Raise(0);
		
	ELSIF fbMcAddAxisToGroup.Done THEN
		eAxesGroupMethodState := AXES_GROUP_METHOD_EXECUTE;
		eAxesGroupState := AXES_GROUP_ADD_DONE;
		
	END_IF
END_CASE
END_METHOD

METHOD PROTECTED MS_AddDone
fbMcAddAxisToGroup( AxesGroup := stAxesGroupRef, Axis := stInternalAxisRef, Execute := FALSE);

IF NOT bAdd THEN
	eAxesGroupState := AXES_GROUP_IDLE;
END_IF
END_METHOD

METHOD PROTECTED MS_GroupDisable
CASE eAxesGroupMethodState OF
	AXES_GROUP_METHOD_EXECUTE:
		fbMcGroupDisable( AxesGroup := stAxesGroupRef, Execute := TRUE);

		IF NOT fbMcGroupDisable.Busy THEN
			eAxesGroupMethodState := AXES_GROUP_METHOD_DONE; 
			
		END_IF
	
	AXES_GROUP_METHOD_DONE:
		IF fbMcGroupDisable.Error THEN
			bError := TRUE;
			iErrorID := fbMcGroupDisable.ErrorID;
			fbMcGroupDisable( AxesGroup := stAxesGroupRef, Execute := FALSE);
		
			fbAlarmGroupDisable.ipArguments.Clear().AddUDInt(iErrorID);
			fbAlarmGroupDisable.Raise(0);
			
		ELSIF fbMcGroupDisable.Done THEN
			eAxesGroupMethodState := AXES_GROUP_METHOD_EXECUTE;
			eAxesGroupState := AXES_GROUP_DISABLE_DONE;	
			
		END_IF
END_CASE
END_METHOD

METHOD PROTECTED MS_GroupDisableDone
fbMcGroupDisable( AxesGroup := stAxesGroupRef, Execute := FALSE);

IF NOT bDisable THEN
	eAxesGroupState := AXES_GROUP_IDLE;
END_IF
END_METHOD

METHOD PROTECTED MS_GroupEnable
CASE eAxesGroupMethodState OF
	AXES_GROUP_METHOD_EXECUTE:
		fbMcGroupEnable( AxesGroup := stAxesGroupRef, Execute := TRUE);
	
		IF NOT fbMcGroupEnable.Busy THEN
			eAxesGroupMethodState := AXES_GROUP_METHOD_DONE; 
			
		END_IF
	
	AXES_GROUP_METHOD_DONE:
		IF fbMcGroupEnable.Error THEN
			bError := TRUE;
			iErrorID := fbMcGroupEnable.ErrorID;
			fbMcGroupEnable( AxesGroup := stAxesGroupRef, Execute := FALSE);
			
			fbAlarmGroupEnable.ipArguments.Clear().AddUDInt(iErrorID);
			fbAlarmGroupEnable.Raise(0);
			
		ELSIF fbMcGroupEnable.Done THEN
			eAxesGroupMethodState := AXES_GROUP_METHOD_EXECUTE;
			eAxesGroupState := AXES_GROUP_ENABLE_DONE;
			
		END_IF
END_CASE
END_METHOD

METHOD PROTECTED MS_GroupEnableDone
fbMcGroupEnable( AxesGroup := stAxesGroupRef, Execute := FALSE);

IF NOT bEnable THEN
	eAxesGroupState := AXES_GROUP_IDLE;
END_IF
END_METHOD

METHOD PROTECTED MS_GroupHalt
VAR
	bFirstCycle : BOOL := TRUE;
END_VAR
CASE eAxesGroupMethodState OF
	AXES_GROUP_METHOD_EXECUTE:
		fbMcGroupHalt( AxesGroup		:= stAxesGroupRef,
						Execute 		:= TRUE,
						Deceleration	:= lrDeceleration,
						Jerk 			:= lrJerk);
			
		IF NOT fbMcGroupHalt.Busy THEN
			eAxesGroupMethodState := AXES_GROUP_METHOD_DONE; 
			
		END_IF
	
	AXES_GROUP_METHOD_DONE:
		IF fbMcGroupHalt.Error THEN
			bError := TRUE;
			iErrorID := fbMcGroupHalt.ErrorID;
			fbMcGroupHalt( AxesGroup := stAxesGroupRef, Execute := FALSE);
			
		ELSIF fbMcGroupHalt.Done THEN
			eAxesGroupMethodState := AXES_GROUP_METHOD_EXECUTE; 
			eAxesGroupState := AXES_GROUP_HALT_DONE;
			
		END_IF
END_CASE
END_METHOD

METHOD PROTECTED MS_GroupHaltDone
VAR_INPUT
END_VAR
fbMcGroupHalt( AxesGroup := stAxesGroupRef, Execute := TRUE);

IF NOT bGroupHalt THEN
	eAxesGroupState := AXES_GROUP_IDLE;
END_IF
END_METHOD

METHOD PROTECTED MS_GroupStop
CASE eAxesGroupMethodState OF
	AXES_GROUP_METHOD_EXECUTE:
		fbMcGroupStop( AxesGroup 		:= stAxesGroupRef,
						Execute 		:= TRUE,
						Deceleration 	:= lrDeceleration,
						Jerk			:= lrJerk);
			
		IF NOT fbMcGroupStop.Busy THEN
			eAxesGroupMethodState := AXES_GROUP_METHOD_DONE; 
			
		END_IF
	
	AXES_GROUP_METHOD_DONE:
		IF fbMcGroupStop.Error THEN
			bError := TRUE;
			iErrorID := fbMcGroupHalt.ErrorID;
			fbMcGroupStop( AxesGroup := stAxesGroupRef, Execute := FALSE);
			
		ELSIF fbMcGroupStop.Done THEN
			eAxesGroupMethodState := AXES_GROUP_METHOD_EXECUTE; 
			eAxesGroupState := AXES_GROUP_STOP_DONE;
			
		END_IF
END_CASE
END_METHOD

METHOD PROTECTED MS_GroupStopDone
VAR_INPUT
END_VAR
IF NOT bGroupStop THEN
	eAxesGroupState := AXES_GROUP_IDLE;
END_IF
END_METHOD

METHOD PROTECTED MS_GroupUnlock
CASE eAxesGroupMethodState OF
	AXES_GROUP_METHOD_EXECUTE:
		fbMcGroupStop( AxesGroup := stAxesGroupRef, Execute := FALSE);
	
		IF NOT fbMcGroupStop.Busy THEN
			eAxesGroupState := AXES_GROUP_UNLOCK_DONE;
			
		END_IF
END_CASE
END_METHOD

METHOD PROTECTED MS_GroupUnlockDone
VAR_INPUT
END_VAR
IF NOT bGroupUnlock THEN
	eAxesGroupState := AXES_GROUP_IDLE;
END_IF
END_METHOD

METHOD PROTECTED MS_Idle
VAR_INPUT
END_VAR
;
END_METHOD

METHOD PROTECTED MS_Initializing
VAR_INPUT
END_VAR
CASE eAxesGroupStateInit OF
	AXES_GROUP_INIT_RESET:
		fbMcGroupReset( AxesGroup := stAxesGroupRef, Execute := TRUE);
			
		IF fbMcGroupReset.Error THEN
			bError := TRUE;
			iErrorID := fbMcGroupReset.ErrorID;
			fbMcGroupReset( AxesGroup := stAxesGroupRef, Execute := FALSE);
	
			fbAlarmGroupReset.ipArguments.Clear().AddUDInt(iErrorID);
			fbAlarmGroupReset.Raise(0);
				
		ELSIF fbMcGroupReset.Done THEN
			fbMcGroupReset( AxesGroup := stAxesGroupRef, Execute := FALSE);
			eAxesGroupStateInit := AXES_GROUP_INIT_ENABLE;	
		END_IF
		
	AXES_GROUP_INIT_ENABLE:
		fbMcGroupEnable( AxesGroup := stAxesGroupRef, Execute := TRUE);
			
		IF fbMcGroupEnable.Error THEN
			bError := TRUE;
			iErrorID := fbMcGroupEnable.ErrorID;
			fbMcGroupEnable( AxesGroup := stAxesGroupRef, Execute := FALSE);
	
			fbAlarmGroupEnable.ipArguments.Clear().AddUDInt(iErrorID);
			fbAlarmGroupEnable.Raise(0);
				
		ELSIF fbMcGroupEnable.Done THEN
			fbMcGroupEnable( AxesGroup := stAxesGroupRef, Execute := FALSE);
			eAxesGroupStateInit := AXES_GROUP_INIT_DONE;	
		END_IF
		
	AXES_GROUP_INIT_DONE:
		IF NOT bInit THEN
			eAxesGroupState := AXES_GROUP_READY_INITIALIZED;
		END_IF
END_CASE
END_METHOD

METHOD PROTECTED MS_ReadyInitialized
VAR_INPUT
END_VAR
eAxesGroupState := AXES_GROUP_IDLE;
END_METHOD

METHOD PROTECTED MS_Remove
CASE eAxesGroupMethodState OF
	AXES_GROUP_METHOD_EXECUTE:
		fbMcRemoveAxisFromGroup(	AxesGroup		:= stAxesGroupRef,
									Execute 		:= TRUE,
									IdentInGroup 	:= UDINT_TO_IDENTINGROUP(iIdentInGroup));
			
		IF NOT fbMcRemoveAxisFromGroup.Busy THEN
			eAxesGroupMethodState := AXES_GROUP_METHOD_DONE; 
			
		END_IF
	
	AXES_GROUP_METHOD_DONE:
		IF fbMcRemoveAxisFromGroup.Error THEN
			bError := TRUE;
			iErrorID := fbMcRemoveAxisFromGroup.ErrorID;
			fbMcRemoveAxisFromGroup(	AxesGroup := stAxesGroupRef,
										Execute := FALSE);
		
			fbAlarmRemoveFromGroup.ipArguments.Clear().AddUDInt(iErrorID);
			fbAlarmRemoveFromGroup.Raise(0);	
		
		ELSIF fbMcRemoveAxisFromGroup.Done THEN
			eAxesGroupMethodState := AXES_GROUP_METHOD_EXECUTE; 
			eAxesGroupState := AXES_GROUP_REMOVE_DONE;
			
		END_IF
END_CASE
END_METHOD

METHOD PROTECTED MS_RemoveAll
CASE eAxesGroupMethodState OF
	AXES_GROUP_METHOD_EXECUTE:
		fbMcUngroupAllAxes( AxesGroup := stAxesGroupRef, Execute := TRUE);
		
	IF NOT fbMcUngroupAllAxes.Busy THEN
		eAxesGroupMethodState := AXES_GROUP_METHOD_DONE; 
		
	END_IF
	
	AXES_GROUP_METHOD_DONE:
	IF fbMcUngroupAllAxes.Error THEN
		bError := TRUE;
		iErrorID := fbMcUngroupAllAxes.ErrorID;
		fbMcUngroupAllAxes( AxesGroup := stAxesGroupRef, Execute := FALSE);
		fbAlarmUngroupAll.ipArguments.Clear().AddUDInt(iErrorID);
		fbAlarmUngroupAll.Raise(0);	
	
	ELSIF bError THEN
		MR_Disable();
		
		IF NOT Busy THEN
			bError := FALSE;
			eAxesGroupMethodState := AXES_GROUP_METHOD_EXECUTE; 
			eAxesGroupState := AXES_GROUP_REMOVE_ALL_DONE;
		END_IF

 	ELSIF fbMcUngroupAllAxes.Done THEN
		eAxesGroupMethodState := AXES_GROUP_METHOD_EXECUTE; 
		eAxesGroupState := AXES_GROUP_REMOVE_ALL_DONE;
		
	END_IF
END_CASE
END_METHOD

METHOD PROTECTED MS_RemoveAllDone
VAR_INPUT
END_VAR
fbMcUngroupAllAxes( AxesGroup := stAxesGroupRef, Execute := FALSE);

IF NOT bRemoveAll THEN
	eAxesGroupState := AXES_GROUP_IDLE;
END_IF
END_METHOD

METHOD PROTECTED MS_RemoveDone
VAR_INPUT
END_VAR
fbMcRemoveAxisFromGroup( AxesGroup := stAxesGroupRef, Execute := FALSE);

IF NOT bRemove THEN
	eAxesGroupState := AXES_GROUP_IDLE;
END_IF
END_METHOD

METHOD PROTECTED MS_Reset
VAR_INPUT
END_VAR
fbMcAddAxisToGroup( AxesGroup := stAxesGroupRef, Axis := stInternalAxisRef, Execute := FALSE);

fbMcRemoveAxisFromGroup( AxesGroup := stAxesGroupRef, Execute := FALSE);

fbMcUngroupAllAxes( AxesGroup := stAxesGroupRef, Execute := FALSE);

fbMcGroupEnable( AxesGroup := stAxesGroupRef, Execute := FALSE);

fbMcGroupDisable( AxesGroup := stAxesGroupRef, Execute := FALSE);

fbMcGroupReadStatus( AxesGroup := stAxesGroupRef, Enable := FALSE);

fbMcGroupReadError( AxesGroup := stAxesGroupRef, Enable := FALSE);
		
fbMcGroupReset( AxesGroup := stAxesGroupRef, Execute := FALSE);

fbMcGroupHalt( AxesGroup := stAxesGroupRef, Execute := FALSE);

fbMcGroupStop( AxesGroup := stAxesGroupRef, Execute := FALSE);

(* Confirming and resetting alarms *)
fbAlarmGroupReset.Confirm( nTimeStamp := 0);
fbAlarmUngroupAll.Confirm( nTimeStamp := 0);
fbAlarmGroupDisable.Confirm( nTimeStamp := 0);
fbAlarmAddAxisToGroup.Confirm( nTimeStamp := 0);
fbAlarmGroupEnable.Confirm( nTimeStamp := 0);
fbAlarmRemoveFromGroup.Confirm( nTimeStamp := 0);

fbAlarmGroupReset.Clear( nTimeStamp := 0, bResetConfirmation := bResetConfirmation); 
fbAlarmUngroupAll.Clear( nTimeStamp := 0, bResetConfirmation := bResetConfirmation); 
fbAlarmGroupDisable.Clear( nTimeStamp := 0, bResetConfirmation := bResetConfirmation); 
fbAlarmAddAxisToGroup.Clear( nTimeStamp := 0, bResetConfirmation := bResetConfirmation); 
fbAlarmGroupEnable.Clear( nTimeStamp := 0, bResetConfirmation := bResetConfirmation); 
fbAlarmRemoveFromGroup.Clear( nTimeStamp := 0, bResetConfirmation := bResetConfirmation); 

IF NOT fbMcGroupStop.Busy THEN
	bGroupLocked := FALSE;
	fbMcGroupReset( AxesGroup := stAxesGroupRef, Execute := TRUE);
	
	IF NOT fbMcGroupReset.Error THEN
		bError := TRUE;
		iErrorID := fbMcGroupReset.ErrorID;
		fbMcGroupReset( AxesGroup := stAxesGroupRef, Execute := FALSE);

		fbAlarmGroupReset.ipArguments.Clear().AddUDInt(iErrorID);
		fbAlarmGroupReset.Raise(0);		

	ELSIF fbMcGroupReset.Done THEN
		eAxesGroupState := AXES_GROUP_RESET_DONE;
		
	END_IF
	
END_IF
END_METHOD

METHOD PROTECTED MS_ResetDone
VAR_INPUT
END_VAR
fbMcGroupReset( AxesGroup := stAxesGroupRef, Execute := FALSE);

IF NOT bReset THEN
	eAxesGroupState := AXES_GROUP_IDLE;
	
END_IF
END_METHOD

METHOD PROTECTED MS_Uninitialized
VAR_INPUT
END_VAR
(* Reset commands *)
bAbort 		:= FALSE;
bReset 		:= FALSE;
bAdd 		:= FALSE;
bRemove 	:= FALSE;
bRemoveAll 	:= FALSE;
bEnable 	:= FALSE;
bDisable 	:= FALSE;
bGroupStop 	:= FALSE;
bGroupHalt 	:= FALSE;
bGroupUnlock:= FALSE;

(* Reset status flags *)
bActive					:= FALSE;
bBusy					:= FALSE;
bError 					:= FALSE;
iErrorID 				:= 0;
eAxesGroupStateInit		:= AXES_GROUP_INIT_RESET;
eAxesGroupStateAbort	:= AXES_GROUP_ABORTING_RESET_FBS;
bAxisAdded				:= FALSE;
bAxisRemoved			:= FALSE;
bRemovedAll				:= FALSE;
bGroupEnabled			:= FALSE;
iAxesInGroup			:= 0;
bGroupLocked			:= FALSE;
END_METHOD

(* Axes group name for other utilities *)
PROPERTY Name : STRING
GET
Name := sName;
END_GET
SET
sName := Name;
END_SET
END_PROPERTY

PROPERTY RemovedAll : REFERENCE TO BOOL
GET
RemovedAll REF= bRemovedAll;
END_GET
END_PROPERTY

PROPERTY State : REFERENCE TO E_AxesGroupCAState
GET
State REF= eAxesGroupState;
END_GET
END_PROPERTY

METHOD PROTECTED StateMachine
VAR_INPUT
END_VAR
CASE eAxesGroupState OF
	AXES_GROUP_UNINITIALIZED:
		MS_Uninitialized();
		
	AXES_GROUP_INITIALIZING:
		MS_Initializing();
	
	AXES_GROUP_READY_INITIALIZED:
		MS_ReadyInitialized();
	
	AXES_GROUP_IDLE:
		MS_Idle();
		
	AXES_GROUP_ADD:
		MS_Add();
		
	AXES_GROUP_ADD_DONE:
		MS_AddDone();
		
	AXES_GROUP_REMOVE:
		MS_Remove();
		
	AXES_GROUP_REMOVE_DONE:
		MS_RemoveDone();
		
	AXES_GROUP_REMOVE_ALL:
		MS_RemoveAll();
		
	AXES_GROUP_REMOVE_ALL_DONE:
		MS_RemoveAllDone();
		
	AXES_GROUP_ENABLE:
		MS_GroupEnable();
		
	AXES_GROUP_ENABLE_DONE:
		MS_GroupEnableDone();
	
	AXES_GROUP_DISABLE:
		MS_GroupDisable();
		
	AXES_GROUP_DISABLE_DONE:
		MS_GroupDisableDone();
		
	AXES_GROUP_RESET:
		MS_Reset();
		
	AXES_GROUP_RESET_DONE:
		MS_ResetDone();
	
	AXES_GROUP_HALT:
		MS_GroupHalt();
		
	AXES_GROUP_HALT_DONE:
		MS_GroupHaltDone();
		
	AXES_GROUP_STOP:
		MS_GroupStop();
		
	AXES_GROUP_STOP_DONE:
		MS_GroupStopDone();
		
	AXES_GROUP_UNLOCK:
		MS_GroupUnlock();
		
	AXES_GROUP_UNLOCK_DONE:
		MS_GroupUnlockDone();
	
	AXES_GROUP_ABORTING:
		MS_Aborting();
		
END_CASE
END_METHOD

PROPERTY StatePlcOpen : REFERENCE TO E_AxesGroupCAStatePlcOpen
GET
StatePlcOpen REF= eStatePlcOpen;
END_GET
END_PROPERTY

END_FUNCTION_BLOCK

// ---- POUs/Axis/FB_AxisServo.TcPOU
(* 
:Description: This function block is used represent basic axis controled by standard PLCopen motion function blocks.
*)
FUNCTION_BLOCK FB_AxisServo EXTENDS FB_UniversalAxis
VAR
	(* MC_Home *)
	eHomingMode		: MC_HomingMode;		(*  *)
	stHomingOptions	: ST_HomingOptions;		(*  *)
	fbMcHome		: MC_Home;				(*  *)
	
	(* Home switch cam *)
	piHomeSwitch	: FB_DigitalInput;		(*  *)
END_VAR

(* Run home switch FB *)
piHomeSwitch();

(* Run parent implementation *)
SUPER^();

PROPERTY HomingMode : MC_HomingMode
GET
HomingMode := eHomingMode;
END_GET
SET
eHomingMode := HomingMode;
END_SET
END_PROPERTY

PROPERTY HomingOptions : ST_HomingOptions
GET
HomingOptions := stHomingOptions;
END_GET
SET
stHomingOptions := HomingOptions;
END_SET
END_PROPERTY

METHOD MR_FirstCycle
VAR_INPUT
	sName 				: STRING; 	(* Axis object name *)
	sMeasurementUnits	: STRING;	(* Measurement units used by axis *)
	bModulo				: BOOL;		(* Axis is periodic *)
END_VAR
SUPER^.MR_FirstCycle(sName:=sName, sMeasurementUnits := sMeasurementUnits, bModulo := bModulo);
piHomeSwitch.MR_FirstCycle(CONCAT(THIS^.sName,', home switch'), sModuleType := piHomeSwitch.ModuleType, sPortID := piHomeSwitch.PortID);
END_METHOD

METHOD PROTECTED MS_Aborting
VAR_INPUT
END_VAR
fbMcHome(Axis := stAxisRef, Execute := FALSE);

SUPER^.MS_Aborting();
END_METHOD

METHOD PROTECTED MS_Halt
VAR_INPUT
END_VAR
(* Reset MC_Home *)
fbMcHome(Axis := stAxisRef, Execute := FALSE);

(* Run parent halt state *)
SUPER^.MS_Halt();
END_METHOD

METHOD PROTECTED MS_Home
VAR_INPUT
END_VAR
fbMcHome(	Axis 			:= stAxisRef,
			Execute 		:= TRUE,
			Position 		:= lrHomePosition,
			HomingMode		:= eHomingMode,
			BufferMode		:= eBufferMode,
			Options			:= stHomingOptions,
			bCalibrationCam := piHomeSwitch.In);
	
IF fbMcHome.Error THEN
	bError := TRUE;
	iErrorID := fbMcHome.ErrorID;
	fbMcHome( Axis := stAxisRef, Execute := FALSE);
	fbAlarmHome.ipArguments.Clear().AddUDInt(iErrorID);	
	fbAlarmHome.Raise(0);
	
ELSIF fbMcHome.Done THEN
	eAxisState := AXIS_HOME_DONE;
		
END_IF
END_METHOD

METHOD PROTECTED MS_HomeDone
VAR_INPUT
END_VAR
fbMcHome(Axis := stAxisRef, Execute := FALSE);

IF NOT bHome AND NOT fbMcHome.Busy THEN
	eAxisState := AXIS_IDLE;
	
END_IF
END_METHOD

METHOD PROTECTED MS_Reset
VAR_INPUT
END_VAR
(* Reset MC_Home*)
fbMcHome( Axis := stAxisRef, Execute := FALSE);

(* Run parent reset procedure*)
IF NOT fbMcHome.Busy THEN
	SUPER^.MS_Reset();
	
END_IF
END_METHOD

METHOD PROTECTED MS_Stop
VAR_INPUT
END_VAR
(* Reset MC_Home *)
fbMcHome(Axis := stAxisRef, Execute := FALSE);

(* Run parent stop state *)
SUPER^.MS_Stop();
END_METHOD

PROPERTY ref_HomeSwitch : REFERENCE TO FB_DigitalInput
GET
ref_HomeSwitch REF= piHomeSwitch;
END_GET
END_PROPERTY

END_FUNCTION_BLOCK

// ---- POUs/Axis/FB_UniversalAxis.TcPOU
(* 
:Description: This function block is base for all other axis devices. It's abstract so it can't be used to create instances.
*)
FUNCTION_BLOCK ABSTRACT FB_UniversalAxis IMPLEMENTS I_UniversalAxis
VAR
	(* Generic *)
	bFirstCycle				: BOOL := TRUE;					(* First cycle bit *)
	sName 					: STRING;						(* Axis name for other utilities *)
	sUnit 					: STRING;						(* Measurement units *)
	bModulo					: BOOL;							(* Axis is periodic *)
	
	(* Hardware link *)
	stAxisRef				: AXIS_REF;						(* Axis reference object *)
	
	(* Internal commands *)
	bInit					: BOOL;							(* Power on axis and prepare to work *)
	bAbort					: BOOL;							(* Power off axis and reset status flags *)
	bHome					: BOOL;							(* Home to reference point *)
	bMoveVelocity			: BOOL;							(* Start motion with constant velocity *)
	bMoveAbsolute			: BOOL;							(* Move to absolute position *)
	bMoveAdditive			: BOOL;							(* Move by distance *)
	bMoveRelative			: BOOL;							(* Move by distance *)
	bJog					: BOOL;							(* Start manual jog movement *)
	bStop					: BOOL;							(* High priority stop command *)
	bHalt					: BOOL;							(* Halt current motion, next motion command will abort this command *)
	bReset					: BOOL;							(* Reset axis and return to READY state *)
	bUnlock					: BOOL;							(* Unlock axis after stop command *)
	//bCouple				: BOOL;							(* Couple appended slave axis *)
	//bDecouple				: BOOL;							(* Decouple appended slave axis *)
	
	(* Internal status - flags *)
	bActive					: BOOL;
	bBusy					: BOOL;							(* Function block currently executes one of the requests *)
	bError					: BOOL;							(* Error status flag *)
	iErrorID				: UDINT;						(* Error ID *)
	iAxisErrorID			: UDINT;						(* Axis error ID *)
	lrActualPosition		: LREAL;						(* Actual axis position in selected units *)
	lrActualVelocity		: LREAL;						(* Actual axis velocity in selected units *)
	bPowerOn 				: BOOL;							(* Power On status bit *)
	bIsHomed				: BOOL;							(* Axis has been homed even once *)
	bInVelocity				: BOOL;							(* Axis is moving in target velocity *)
	bInPostion				: BOOL;							(* Axis reached target position *)
	bMoveActive				: BOOL;							(* Axis is moving to target position *)
	bJogDone				: BOOL;							(* Axis manual movement by jog done *)
	bStopped				: BOOL;							(* Axis movement has been stopped *)
	bHalted					: BOOL;							(* Axis movement has been halted *)
	bLocked					: BOOL;							(* Axis locked after stop commad *)
	eStatePlcOpen			: E_AxisStatePlcOpen;			(* Current PLCOpen state of axis *)
	bHaltLog 				: BOOL;							(* Halt request flag for machine logger *)
	bStopLog 				: BOOL;							(* Stop request flag for machine logger *)
	
	(* Internal status - state machines *)
	eAxisState 				: E_AxisState;					(* Main axis state machine *)
	eAxisStateBeforeReset 	: E_AxisState;					(* State before reset command *)
	eAxisStateInit 			: E_AxisStateInit;				(* Init axis state machine *)
	
	(* General parameters *)
	lrOverride				: LREAL;						(* Axis velocity override in percents [%] *)
	lrVelocity 				: LREAL;						(* Axis velocity in measurement units per second *)
	lrAcceleration			: LREAL;						(* Axis acceleration in measurement units per sercond^2 *)
	lrDeceleration 			: LREAL;						(* Axis deceleration in measurement units per sercond^2 *)
	lrJerk					: LREAL;						(* Axis jerk in measurement unit per sercond^3 *)
	lrAbsolutePosition		: LREAL;						(* Target position for MC_MoveAbsolute function *)
	lrRelativeDistance		: LREAL;						(* Relative distance to move for MC_MoveRelative/Additive fuctions *)
	lrHomePosition			: LREAL;						(* This parameters is used to set axis position while performing homing procedure *)
	
	(* Jog function parameters *)	
	bJogActive				: BOOL;
	lrJogPosition			: LREAL;						(* Relative position to move for jog feature *)
	lrJogVelocity			: LREAL;						(* Jog movement velocity *)
	lrJogAcceleration		: LREAL;						(* Jog movement acceleration *)
	lrJogDeceleration		: LREAL;						(* Jog movement deceleration *)
	lrJogJerk				: LREAL;						(* Jog movement jerk *)
	eJogMode				: E_JogMode;					(* Jog momement mode *)
	eJogDirection			: E_AxisJogDirection;			(* Direction of jog movement *)
	
	(* Stop function parameters *)
	lrStopDeceleration		: LREAL;						(* Stop deceleration *)
	lrStopJerk 				: LREAL;						(* Stop jerk *)
	
	(* Other parameters *)
	stOptions				: ST_MoveOptions;				(* Additional movement options *)
	eDirection				: Tc2_MC2.MC_Direction;			(* Axis movement direction for MC_MoveVelocity *)
	eBufferMode 			: MC_BufferMode := MC_Aborting;	(* Axis buffering mode *)
	
	(* Function blocks - readers *)
	fbReadActualPostion		: MC_ReadActualPosition;		(* FB to read actual position *)
	fbReadActualVelocity	: MC_ReadActualVelocity;		(* FB to read actual velocity *)
	fbReadAxisError			: MC_ReadAxisError;				(* FB to read axis error *)
	fbReadAxisStatus	 	: MC_ReadStatus;				(* FB to read axis status *)
	
	(* Function blocks - administrative *)
	fbMcPower				: MC_Power;						(* FB to control axis power supply and override parameter *)
	fbMcReset				: MC_Reset;						(* FB to reset axis errors *)
	
	(* Function blocks - motion *)
	fbMcMoveVelocity		: MC_MoveVelocity;				(* FB to move axis with constant velocity *)
	fbMcMoveAbsolute		: MC_MoveAbsolute;				(* FB to move axis to absolute postion *)
	fbMcMoveAdditive		: MC_MoveAdditive;				(* FB to move axis by relative distance *)
	fbMcMoveRelative		: MC_MoveRelative;				(* FB to move axis by relative distance *)
	fbMcJog 				: MC_Jog;						(* FB to start axis jog movement *)
	fbMcStop				: MC_Stop;						(* FB to stop axis *)
	fbMcHalt				: MC_Halt;						(* FB to halt axis movement *)
	
	(* Function blocks - linear coupling *)
	fbMcGearIn				: MC_GearIn;					(* FB to couple axis *)		
	fbMcGearOut				: MC_GearOut;					(* FB to decouple axis *)
	
	(* Tc3 EventLogger - messages *)
	fbAlarmHalt 			: FB_TcAlarm;				(*  *)
	fbAlarmInitReset		: FB_TcAlarm;				(*  *)
	fbAlarmInitPowerOn		: FB_TcAlarm;				(*  *)
	fbAlarmMoveAbsolute		: FB_TcAlarm;				(*  *)
	fbAlarmMoveAdditive		: FB_TcAlarm;				(*  *)
	fbAlarmMoveJog			: FB_TcAlarm;				(*  *)	
	fbAlarmMoveRelative		: FB_TcAlarm;				(*  *)	
	fbAlarmMoveVelocity		: FB_TcAlarm;				(*  *)	
	fbAlarmStop				: FB_TcAlarm;				(*  *)
	fbAlarmHome				: FB_TcAlarm;				(*  *)	
	
	fbAlarmHaltCA			: FB_TcAlarm;				(*  *)	
	fbAlarmMoveAbsoluteCA	: FB_TcAlarm;				(*  *)
	fbAlarmMoveRelativeCA	: FB_TcAlarm;				(*  *)
	
	fbAlarmCoupling			: FB_TcAlarm;				(*  *)
	fbAlarmDecoupling		: FB_TcAlarm;				(*  *)		

	bResetConfirmation 		: BOOL;						(*  *)	
	
	rtError					: R_TRIG; 					(* Rising edge trigger for function block error *)

END_VAR

(* Run first cycle procedure *)
IF bFirstCycle THEN
	bFirstCycle := FALSE;
		
	fbAlarmHalt.CreateEx( 	stEventEntry := TC_EVENTS.ShellAxisEventClass.Halt, 
							bWithConfirmation := 1,
							ipSourceInfo := 0);
									
	fbAlarmInitReset.CreateEx( 	stEventEntry := TC_EVENTS.ShellAxisEventClass.InitReset, 
								bWithConfirmation := 1,
								ipSourceInfo := 0);
		
	fbAlarmInitPowerOn.CreateEx( 	stEventEntry := TC_EVENTS.ShellAxisEventClass.InitPowerOn, 
									bWithConfirmation := 1,
									ipSourceInfo := 0);
									
	fbAlarmMoveAbsolute.CreateEx( 	stEventEntry := TC_EVENTS.ShellAxisEventClass.MoveAbsolute, 
									bWithConfirmation := 1,
									ipSourceInfo := 0);
		
	fbAlarmMoveAdditive.CreateEx(	stEventEntry := TC_EVENTS.ShellAxisEventClass.MoveAdditive, 
									bWithConfirmation := 1,
									ipSourceInfo := 0);
									
	fbAlarmMoveJog.CreateEx( 	stEventEntry := TC_EVENTS.ShellAxisEventClass.MoveJog, 
								bWithConfirmation := 1,
								ipSourceInfo := 0);
		
	fbAlarmMoveRelative.CreateEx( stEventEntry := TC_EVENTS.ShellAxisEventClass.MoveRelative, 
									bWithConfirmation := 1,
									ipSourceInfo := 0);
									
	fbAlarmMoveVelocity.CreateEx(	stEventEntry := TC_EVENTS.ShellAxisEventClass.MoveVelocity, 
									bWithConfirmation := 1,
									ipSourceInfo := 0);
		
	fbAlarmStop.CreateEx( 	stEventEntry := TC_EVENTS.ShellAxisEventClass.Stop, 
							bWithConfirmation := 1,
							ipSourceInfo := 0);
									
	fbAlarmHome.CreateEx( 	stEventEntry := TC_EVENTS.ShellAxisEventClass.Home, 
							bWithConfirmation := 1,
							ipSourceInfo := 0);									

	fbAlarmHaltCA.CreateEx( stEventEntry := TC_EVENTS.ShellAxisEventClass.HaltCA, 
							bWithConfirmation := 1,
							ipSourceInfo := 0);
		
	fbAlarmMoveAbsoluteCA.CreateEx( stEventEntry := TC_EVENTS.ShellAxisEventClass.MoveAbsoluteCA, 
									bWithConfirmation := 1,
									ipSourceInfo := 0);
									
	fbAlarmMoveRelativeCA.CreateEx( stEventEntry := TC_EVENTS.ShellAxisEventClass.MoveRelativeCA, 
									bWithConfirmation := 1,
									ipSourceInfo := 0);
		
	fbAlarmCoupling.CreateEx( stEventEntry := TC_EVENTS.ShellAxisEventClass.Coupling, 
									bWithConfirmation := 1,
									ipSourceInfo := 0);
									
	fbAlarmDecoupling.CreateEx( stEventEntry := TC_EVENTS.ShellAxisEventClass.Decoupling, 
									bWithConfirmation := 1,
									ipSourceInfo := 0);									
									
END_IF

(* Read AXIS_REF status *)
stAxisRef.ReadStatus();

(* Read axis PLCOpen state *)
fbReadAxisStatus( Axis := stAxisRef, Enable := TRUE);
					
IF fbReadAxisStatus.Valid THEN
	IF fbReadAxisStatus.Disabled THEN
		eStatePlcOpen := AXIS_PLCOPEN_DISABLED;
		
	ELSIF fbReadAxisStatus.StandStill THEN
		eStatePlcOpen := AXIS_PLCOPEN_STANDSTILL;
		
	ELSIF fbReadAxisStatus.Homing THEN
		eStatePlcOpen := AXIS_PLCOPEN_HOMING;
		
	ELSIF fbReadAxisStatus.DiscreteMotion THEN
		eStatePlcOpen := AXIS_PLCOPEN_DISCRETE_MOTION;
		
	ELSIF fbReadAxisStatus.ContinuousMotion THEN
		eStatePlcOpen := AXIS_PLCOPEN_CONTINUOUS_MOTION;
		
	ELSIF fbReadAxisStatus.SynchronizedMotion THEN
		eStatePlcOpen := AXIS_PLCOPEN_SYNCHRONIZED_MOTION;
		
	ELSIF fbReadAxisStatus.ErrorStop THEN
		eStatePlcOpen := AXIS_PLCOPEN_ERRORSTOP;
		
	END_IF
END_IF

(* Update status flags *)
bActive := (eAxisState >= AXIS_READY_INITIALIZED);
bBusy := eAxisState <> AXIS_UNINITIALIZED AND eAxisState <> AXIS_IDLE;
bPowerOn := NOT stAxisRef.Status.Disabled;

(* Read axis errors *)
fbReadAxisError(	Axis := stAxisRef,
					Enable := TRUE,
					AxisErrorID => iAxisErrorID);

(* Read actual axis postion *)
IF bModulo THEN
	lrActualPosition := stAxisRef.NcToPlc.ModuloActPos;
ELSE
	fbReadActualPostion(	Axis := stAxisRef,
							Enable := TRUE,
							Position => lrActualPosition);
END_IF


(* Read actual axis velocity *)
fbReadActualVelocity( 	Axis := stAxisRef,
						Enable := TRUE,
						ActualVelocity => lrActualVelocity);		

(* Report errors that occur *)
rtError(CLK:=bError);

IF rtError.Q THEN 
	fbMachineLogger.MR_AddLogs(FUN_MergeStrings5(sName, ' : Error occured (error ID: ', UDINT_TO_STRING(iErrorID), ')', ''));

END_IF
						
(* Execute main state machine *)
StateMachine();

PROPERTY Acceleration : LREAL
GET
Acceleration := lrAcceleration;
END_GET
SET
lrAcceleration := Acceleration;
END_SET
END_PROPERTY

PROPERTY Active : REFERENCE TO BOOL
GET
Active REF= bActive;
END_GET
END_PROPERTY

PROPERTY ActualPosition : REFERENCE TO LREAL
GET
ActualPosition REF= lrActualPosition;
END_GET
END_PROPERTY

PROPERTY ActualVelocity : REFERENCE TO LREAL
GET
ActualVelocity REF= lrActualVelocity;
END_GET
END_PROPERTY

PROPERTY AxisErrorID : REFERENCE TO UDINT
GET
AxisErrorID REF= iAxisErrorID;
END_GET
END_PROPERTY

PROPERTY AxisRef : AXIS_REF
GET
AxisRef := stAxisRef;
END_GET
SET
stAxisRef := AxisRef;
END_SET
END_PROPERTY

PROPERTY BufferMode : Tc2_MC2.MC_BufferMode
GET
BufferMode := eBufferMode;
END_GET
SET
eBufferMode := BufferMode;
END_SET
END_PROPERTY

PROPERTY Busy : REFERENCE TO BOOL
GET
Busy REF= bBusy;
END_GET
END_PROPERTY

PROPERTY Coupled : REFERENCE TO BOOL
GET
END_GET
END_PROPERTY

PROPERTY Deceleration : LREAL
GET
Deceleration := lrDeceleration;
END_GET
SET
lrDeceleration := Deceleration;
END_SET
END_PROPERTY

PROPERTY Direction : Tc2_MC2.MC_Direction
GET
Direction := eDirection;
END_GET
SET
eDirection := Direction;
END_SET
END_PROPERTY

PROPERTY Error : REFERENCE TO BOOL
GET
Error REF= bError;
END_GET
END_PROPERTY

PROPERTY ErrorID : REFERENCE TO UDINT
GET
ErrorID REF= iErrorID;
END_GET
END_PROPERTY

PROPERTY Halted : REFERENCE TO BOOL
GET
Halted REF= bHalted;
END_GET
END_PROPERTY

PROPERTY InPosition : REFERENCE TO BOOL
GET
InPosition REF= bInPostion;
END_GET
END_PROPERTY

PROPERTY InVelocity : REFERENCE TO BOOL
GET
InVelocity REF= bInVelocity;
END_GET
END_PROPERTY

PROPERTY IsHomed : REFERENCE TO BOOL
GET
IsHomed REF= bIsHomed;
END_GET
END_PROPERTY

PROPERTY Jerk : LREAL
GET
Jerk := lrJerk;
END_GET
SET
lrJerk := Jerk;
END_SET
END_PROPERTY

PROPERTY JogAcceleration : LREAL
GET
JogAcceleration := lrJogAcceleration;
END_GET
SET
lrJogAcceleration := JogAcceleration;
END_SET
END_PROPERTY

PROPERTY JogDeceleration : LREAL
GET
JogDeceleration := lrJogDeceleration;
END_GET
SET
lrJogDeceleration := JogDeceleration;
END_SET
END_PROPERTY

PROPERTY JogDirection : E_AxisJogDirection
GET
JogDirection := eJogDirection;
END_GET
SET
eJogDirection := JogDirection;
END_SET
END_PROPERTY

PROPERTY JogDone : REFERENCE TO BOOL
GET
JogDone REF= bJogDone;
END_GET
END_PROPERTY

PROPERTY JogJerk : LREAL
GET
JogJerk := lrJogJerk;
END_GET
SET
lrJogJerk := JogJerk;
END_SET
END_PROPERTY

PROPERTY JogMode : Tc2_MC2.E_JogMode
GET
JogMode := eJogMode;
END_GET
SET
eJogMode := JogMode;
END_SET
END_PROPERTY

PROPERTY JogPosition : LREAL
GET
JogPosition := lrJogPosition;
END_GET
SET
lrJogPosition := JogPosition;
END_SET
END_PROPERTY

PROPERTY JogVelocity : LREAL
GET
JogVelocity := lrJogVelocity;
END_GET
SET
lrJogVelocity := JogVelocity;
END_SET
END_PROPERTY

PROPERTY LagError : LREAL
GET
LagError := stAxisRef.NcToPlc.PosDiff;
END_GET
END_PROPERTY

PROPERTY Locked : REFERENCE TO BOOL
GET
Locked REF= bLocked;
END_GET
END_PROPERTY

PROPERTY MoveActive : REFERENCE TO BOOL
GET
MoveActive REF= bMoveActive;
END_GET
END_PROPERTY

METHOD MR_Abort : BOOL
IF eAxisState >= AXIS_INITIALIZING THEN
	bAbort := TRUE;
	eAxisState := AXIS_ABORTING;
	fbMachineLogger.MR_AddLogs(CONCAT(sName,' : abort requested'));
	
ELSIF eAxisState = AXIS_UNINITIALIZED THEN
	bAbort 		:= FALSE;
	MR_Abort	:= TRUE;
	fbMachineLogger.MR_AddLogs(CONCAT(sName,' : abort done'));
	
END_IF
END_METHOD

METHOD MR_Couple : BOOL
VAR_INPUT
END_VAR
;
END_METHOD

METHOD MR_Decouple : BOOL
VAR_INPUT
END_VAR
;
END_METHOD

METHOD MR_FirstCycle
VAR_INPUT
	sName 				: STRING; 	(* Axis object name *)
	sMeasurementUnits	: STRING;	(* Measurement units used by axis *)
	bModulo				: BOOL;		(* Axis is periodic *)
END_VAR
THIS^.sName := sName;
THIS^.sUnit := sMeasurementUnits;
THIS^.bModulo := bModulo;
END_METHOD

METHOD MR_Halt : BOOL
IF eAxisState >= AXIS_IDLE AND eAxisState <> AXIS_HALT_DONE THEN
	IF NOT bHaltLog THEN 
		fbMachineLogger.MR_AddLogs(CONCAT(sName,' : halt requested'));
		bHaltLog := TRUE;
	END_IF
	
	bHalt := TRUE;
	eAxisState := AXIS_HALT;
	
ELSIF eAxisState = AXIS_HALT_DONE THEN
	bInPostion 	:= FALSE;
	bInVelocity := FALSE;
	bMoveActive := FALSE;
	bStopped 	:= FALSE;
	bHalted 	:= TRUE;
	bJogDone 	:= FALSE;
	
	bHalt		:= FALSE;
	MR_Halt 	:= TRUE;

	bHaltLog 	:= FALSE;
	fbMachineLogger.MR_AddLogs(CONCAT(sName,' : halt done'));
	
END_IF
END_METHOD

METHOD MR_Home : BOOL
VAR_INPUT
	lrHomePosition : LREAL;
END_VAR
IF eAxisState = AXIS_IDLE THEN
	THIS^.lrHomePosition := lrHomePosition;
	bIsHomed := FALSE;
	
	bHome := TRUE;
	eAxisState := AXIS_HOME;
	fbMachineLogger.MR_AddLogs(CONCAT(sName,' : home position requested'));
	
ELSIF eAxisState = AXIS_HOME_DONE THEN
	bIsHomed := TRUE;
	
	bHome := FALSE;
	MR_Home := TRUE;
	fbMachineLogger.MR_AddLogs(CONCAT(sName,' : home position done'));	
	
END_IF
END_METHOD

METHOD MR_Init : BOOL
IF eAxisState = AXIS_UNINITIALIZED THEN
	bInit := TRUE;
	fbMachineLogger.MR_AddLogs(CONCAT(sName,' : initialization requested'));
	
ELSIF eAxisState = AXIS_INITIALIZING AND eAxisStateInit = AXIS_INIT_DONE THEN
	//bPowerOn 	:= TRUE;
	bInPostion 	:= FALSE;
	bInVelocity := FALSE;
	bMoveActive := FALSE;
	bStopped 	:= FALSE;
	bHalted 	:= FALSE;
	bJogDone 	:= FALSE;

	bInit 		:= FALSE;
	MR_Init 	:= TRUE;
	
	fbMachineLogger.MR_AddLogs(CONCAT(sName,' : initialization done'));

END_IF
END_METHOD

METHOD MR_Jog : BOOL
VAR_INPUT
	bJogActive	  : BOOL;
END_VAR
THIS^.bJogActive := bJogActive;

IF eAxisState = AXIS_IDLE THEN
	bJog := TRUE;
	bInPostion 	:= FALSE;
	bInVelocity	:= FALSE;
	bMoveActive	:= TRUE;
	bStopped	:= FALSE;
	bHalted 	:= FALSE;
	bJogDone 	:= FALSE;
	
	eAxisState := AXIS_MOVE_JOG;
	fbMachineLogger.MR_AddLogs(CONCAT(sName,' : move jog requested'));	
	
ELSIF eAxisState = AXIS_MOVE_JOG_DONE THEN
	IF eJogMode = E_JogMode.MC_JOGMODE_INCHING OR eJogMode = E_JogMode.MC_JOGMODE_INCHING_MODULO THEN
		bInPostion 	:= TRUE;
	END_IF
	
	bInVelocity := FALSE;
	bMoveActive := FALSE;
	bStopped 	:= FALSE;
	bHalted 	:= FALSE;
	bJogDone 	:= TRUE;	

	bJog 		:= FALSE;
	MR_Jog 		:= TRUE;
	
	fbMachineLogger.MR_AddLogs(CONCAT(sName,' : move jog done'));		
	
END_IF
END_METHOD

METHOD MR_MoveAbsolute : BOOL
VAR_INPUT
	lrAbsolutePosition : LREAL;
END_VAR
IF eAxisState = AXIS_IDLE AND THIS^.lrActualPosition <> lrAbsolutePosition THEN
	THIS^.lrAbsolutePosition := lrAbsolutePosition;
	bMoveAbsolute := TRUE;
	bInPostion 	:= FALSE;
	bInVelocity := FALSE;
	bMoveActive := TRUE;
	bStopped 	:= FALSE;
	bHalted 	:= FALSE;
	bJogDone 	:= FALSE;
	
	eAxisState := AXIS_MOVE_ABSOLUTE;
	fbMachineLogger.MR_AddLogs(CONCAT(sName,' : move absolute requested'));		
	
ELSIF eAxisState = AXIS_MOVE_ABSOLUTE_DONE THEN
	bInPostion 		:= TRUE;
	bInVelocity		:= FALSE;
	bMoveActive 	:= FALSE;
	bStopped 		:= FALSE;
	bHalted			:= FALSE;
	bJogDone 		:= FALSE;
	
	bMoveAbsolute 	:= FALSE;
	MR_MoveAbsolute := TRUE;
	fbMachineLogger.MR_AddLogs(CONCAT(sName,' : move absolute done'));		
	
END_IF
END_METHOD

METHOD MR_MoveAdditive : BOOL
VAR_INPUT
	lrRelativeDistance : LREAL;
END_VAR
THIS^.lrRelativeDistance := lrRelativeDistance;
IF eAxisState = AXIS_IDLE AND THIS^.lrRelativeDistance <> 0.0 THEN
	bMoveAdditive := TRUE;
	bInPostion 	:= FALSE;
	bInVelocity := FALSE;
	bStopped 	:= FALSE;
	bHalted 	:= FALSE;
	bJogDone 	:= FALSE;
	
	bMoveActive := TRUE;
	eAxisState := AXIS_MOVE_ADDITIVE;
	fbMachineLogger.MR_AddLogs(CONCAT(sName,' : move additive requested'));		
	
ELSIF eAxisState = AXIS_MOVE_ADDITIVE_DONE THEN
	bInPostion 		:= TRUE;
	bInVelocity 	:= FALSE;
	bStopped 		:= FALSE;
	bHalted 		:= FALSE;
	bJogDone 		:= FALSE;
	
	bMoveAdditive 	:= FALSE;
	MR_MoveAdditive := TRUE;
	fbMachineLogger.MR_AddLogs(CONCAT(sName,' : move additive done'));		
	
END_IF
END_METHOD

METHOD MR_MoveRelative : BOOL
VAR_INPUT
	lrRelativeDistance : LREAL;
END_VAR
THIS^.lrRelativeDistance := lrRelativeDistance;
IF eAxisState = AXIS_IDLE AND THIS^.lrRelativeDistance <> 0.0 THEN
	bMoveRelative := TRUE;
	bInPostion 	:= FALSE;
	bInVelocity := FALSE;
	bMoveActive := TRUE;
	bStopped 	:= FALSE;
	bHalted 	:= FALSE;
	bJogDone 	:= FALSE;
	
	eAxisState := AXIS_MOVE_RELATIVE;
	fbMachineLogger.MR_AddLogs(CONCAT(sName,' : move relative requested'));			
	
ELSIF eAxisState = AXIS_MOVE_RELATIVE_DONE THEN
	bMoveRelative 	:= FALSE;
	MR_MoveRelative := TRUE;
	
	bInPostion 		:= TRUE;
	bInVelocity 	:= FALSE;
	bMoveActive 	:= FALSE;
	bStopped 		:= FALSE;
	bHalted 		:= FALSE;
	bJogDone 		:= FALSE;
	
	fbMachineLogger.MR_AddLogs(CONCAT(sName,' : move relative done'));		
	
END_IF
END_METHOD

METHOD MR_MoveVelocity : BOOL
IF eAxisState = AXIS_IDLE THEN
	bMoveVelocity 	:= TRUE;
	bInPostion 		:= FALSE;
	bInVelocity 	:= FALSE;
	bMoveActive 	:= TRUE;
	bStopped 		:= FALSE;
	bHalted 		:= FALSE;
	bJogDone 		:= FALSE;	
	
	eAxisState 		:= AXIS_MOVE_VELOCITY;
	fbMachineLogger.MR_AddLogs(CONCAT(sName,' : move velocity requested'));			
	
ELSIF eAxisState = AXIS_MOVE_VELOCITY_DONE THEN
	bMoveVelocity 	:= FALSE;
	MR_MoveVelocity := TRUE;
	
	bInPostion 		:= FALSE;
	bInVelocity 	:= TRUE;
	bMoveActive 	:= TRUE;
	bStopped 		:= FALSE;
	bHalted 		:= FALSE;
	bJogDone 		:= FALSE;
	
	fbMachineLogger.MR_AddLogs(CONCAT(sName,' : move velocity done'));		
	
END_IF
END_METHOD

METHOD MR_Reset : BOOL
IF eAxisState <> AXIS_RESET AND eAxisState <> AXIS_RESET_DONE AND bError THEN
	bReset := TRUE;
	eAxisStateBeforeReset := eAxisState;
	eAxisState := AXIS_RESET;
	fbMachineLogger.MR_AddLogs(CONCAT(sName,' : reset requested'));			
	
ELSIF eAxisState = AXIS_RESET_DONE THEN
	bError := FALSE;
	iErrorID := 0;
	
	bReset := FALSE;
	MR_Reset := TRUE;
	
	fbMachineLogger.MR_AddLogs(CONCAT(sName,' : reset done'));		
		
END_IF
END_METHOD

METHOD MR_Stop : BOOL
IF eAxisState >= AXIS_IDLE AND eAxisState <> AXIS_STOP_DONE THEN
	IF NOT bStopLog THEN 
		fbMachineLogger.MR_AddLogs(CONCAT(sName,' : stop requested'));
		bStopLog := TRUE;	
	END_IF
	
	bStop := TRUE;
	eAxisState := AXIS_STOP;
	
ELSIF eAxisState = AXIS_STOP_DONE THEN
	bStop 		:= FALSE;
	MR_Stop 	:= TRUE;
	
	bInPostion 	:= FALSE;
	bInVelocity := FALSE;
	bMoveActive := FALSE;
	bStopped 	:= TRUE;
	bHalted 	:= FALSE;
	bJogDone 	:= FALSE;
	bLocked		:= TRUE;
	
	bStopLog 	:= FALSE;
	fbMachineLogger.MR_AddLogs(CONCAT(sName,' : stop done'));			
END_IF
END_METHOD

METHOD MR_Unlock : BOOL
VAR_INPUT
END_VAR
IF eAxisState = AXIS_IDLE THEN
	bUnlock := TRUE;
	MR_Unlock := FALSE;
	eAxisState := AXIS_UNLOCK;
	fbMachineLogger.MR_AddLogs(CONCAT(sName,' : unlock after stop requested'));
	
ELSIF eAxisState = AXIS_UNLOCK_DONE THEN
	bUnlock := FALSE;
	MR_Unlock := TRUE;
	bLocked := FALSE;
	fbMachineLogger.MR_AddLogs(CONCAT(sName,' : unlock after stop done'));
	
END_IF
END_METHOD

METHOD PROTECTED MS_Aborting
VAR_INPUT
END_VAR
(* Reset MC_Halt *)
fbMcHalt( Axis := stAxisRef, Execute := FALSE);

(* Reset MC_Stop *)
fbMcStop( Axis := stAxisRef, Execute := FALSE);

(* Reset MC_MoveVelocity *)
fbMcMoveVelocity( Axis := stAxisRef, Execute := FALSE);

(* Reset MC_MoveAbsolute *)
fbMcMoveAbsolute( Axis := stAxisRef, Execute := FALSE);

(* Reset MC_MoveAdditive *)
fbMcMoveAdditive( Axis := stAxisRef, Execute := FALSE);

(* Reset MC_MoveRelative *)
fbMcMoveRelative( Axis := stAxisRef, Execute := FALSE);

(* Reset MC_Jog *)
fbMcJog( Axis := stAxisRef, JogForward := FALSE ,JogBackwards := FALSE);

(* Reset MC_Reset *)
fbMcReset( Axis := stAxisRef, Execute := FALSE);

(* Reset MC_Power *)
fbMcPower(	Enable 			:= FALSE,
			Enable_Positive := FALSE,
			Enable_Negative := FALSE,
			Override 		:= lrOverride,
			Axis 			:= stAxisRef);
					
IF fbReadAxisStatus.Disabled AND NOT fbMcStop.Busy THEN
	bInPostion	:= FALSE;
	bInVelocity := FALSE;
	bMoveActive := FALSE;
	bStopped 	:= FALSE;
	bHalted 	:= FALSE;
	bJogDone	:= FALSE;
	bIsHomed 	:= FALSE;
	bLocked		:= FALSE;
	eAxisState	:= AXIS_UNINITIALIZED;	
	
END_IF
END_METHOD

METHOD PROTECTED MS_Couple : BOOL
VAR_INPUT
END_VAR
(*
IF NOT fbMcGearIn.Error THEN
	fbMcGearIn( Master				:=,
				Slave 				:= ,
				Execute 			:= TRUE,
				RatioNumerator		:=,
				RatioDenominator 	:=,
				Acceleration 		:= ,
				Deceleration 		:= ,
				Jerk 				:=,
				BufferMode 			:=,
				Options				:=);
				
	IF fbMcGearIn.InGear THEN
		eAxisState := AXIS_COUPLE_DONE;
	END_IF
ELSE
	bError := TRUE;
	iErrorID := fbMcGearIn.ErrorID;
	fbMcGearIn( Master := , Slave := , Execute := FALSE);
	fbAlarmCoupling.ipArguments.Clear().AddUDInt(iErrorID);
	fbAlarmCoupling.Raise(0);
END_IF
*)
END_METHOD

METHOD MS_CoupleDone : BOOL
VAR_INPUT
END_VAR
END_METHOD

METHOD MS_Decouple : BOOL
VAR_INPUT
END_VAR
(*
IF NOT fbMcGearOut.Error THEN			
	fbMcGearOut( 	Slave 	:=,
					Execute := TRUE,
					Options := );	
				
	IF fbMcGearOut.Done THEN
		eAxisState := AXIS_DECOUPLE_DONE;
	END_IF
ELSE
	bError := TRUE;
	iErrorID := fbMcGearOut.ErrorID;
	fbMcGearOut( Slave := , Execute := FALSE);
	fbAlarmDecoupling.ipArguments.Clear().AddUDInt(iErrorID);
	fbAlarmDecoupling.Raise(0);
END_IF
*)
END_METHOD

METHOD MS_DecoupleDone : BOOL
VAR_INPUT
END_VAR
END_METHOD

METHOD MS_Extension : BOOL
VAR_INPUT
END_VAR
END_METHOD

METHOD PROTECTED MS_Halt
VAR_INPUT
END_VAR
(* Reset MC_MoveVelocity *)
fbMcMoveVelocity( Axis := stAxisRef, Execute := FALSE);

(* Reset MC_MoveAbsolute *)					
fbMcMoveAbsolute( Axis := stAxisRef, Execute := FALSE);

(* Reset MC_MoveAdditive *)					
fbMcMoveAdditive( Axis := stAxisRef ,Execute := FALSE);

(* Reset MC_MoveRelative *)					
fbMcMoveRelative( Axis := stAxisRef, Execute := FALSE);

(* Reset MC_Jog *)
fbMcJog( Axis := stAxisRef, JogForward := FALSE, JogBackwards := FALSE);

fbMcHalt(	Axis			:= stAxisRef,
			Execute 		:= TRUE,
			Deceleration 	:= lrDeceleration,
			Jerk 			:= lrJerk,
			BufferMode 		:= MC_Aborting);

IF fbMcHalt.Error THEN
	bError := TRUE;
	iErrorID := fbMcHalt.ErrorID;
	fbMcHalt(Axis := stAxisRef, Execute := FALSE);
	fbAlarmHalt.ipArguments.Clear().AddUDInt(iErrorID);
	fbAlarmHalt.Raise(0);

ELSIF fbMcHalt.Done THEN
	eAxisState := AXIS_HALT_DONE;
END_IF
END_METHOD

METHOD PROTECTED MS_HaltDone
VAR_INPUT
END_VAR
fbMcHalt( Axis := stAxisRef, Execute := FALSE);

IF NOT bHalt AND NOT fbMcHalt.Busy THEN
	eAxisState := AXIS_IDLE;
END_IF
END_METHOD

METHOD PROTECTED ABSTRACT MS_Home
VAR_INPUT
END_VAR
END_METHOD

METHOD PROTECTED ABSTRACT MS_HomeDone
VAR_INPUT
END_VAR
END_METHOD

METHOD PROTECTED MS_Idle
VAR_INPUT
END_VAR
;
END_METHOD

METHOD PROTECTED MS_Initializing
VAR_INPUT
END_VAR
CASE eAxisStateInit OF
	AXIS_INIT_RESET:
		fbMcReset(	Execute := TRUE, Axis := stAxisRef);
		
		IF fbMcReset.Error THEN
			bError := fbMcReset.Error;
			iErrorID := fbMcReset.ErrorID;
			fbMcReset(Axis := stAxisRef, Execute := FALSE);
			fbAlarmInitReset.ipArguments.Clear().AddUDInt(iErrorID);
			fbAlarmInitReset.Raise(0);
			
		ELSIF fbMcReset.Done THEN
			fbMcReset(Axis := stAxisRef, Execute := FALSE);
			eAxisStateInit := AXIS_INIT_POWER_ON;
			
		END_IF
		
	AXIS_INIT_POWER_ON:
		fbMcPower(	Enable 			:= TRUE,
					Enable_Positive := TRUE,
					Enable_Negative := TRUE,
					Override 		:= lrOverride,
					Axis 			:= stAxisRef);
			
		IF fbMcPower.Error THEN
			bError := fbMcPower.Error;
			iErrorID := fbMcPower.ErrorID;
			fbAlarmInitPowerOn.ipArguments.Clear().AddUDInt(iErrorID);
			fbAlarmInitPowerOn.Raise(0);			
			
		ELSIF fbMcPower.Status THEN
			eAxisStateInit := AXIS_INIT_DONE;	
				
		END_IF
	
	AXIS_INIT_DONE:
		IF NOT bInit THEN
			eAxisState := AXIS_READY_INITIALIZED;
		END_IF
END_CASE
END_METHOD

METHOD PROTECTED MS_MoveAbsolute
VAR_INPUT
END_VAR
fbMcMoveAbsolute(	Axis			:= stAxisRef,
					Execute 		:= TRUE,
					Position 		:= lrAbsolutePosition,
					Velocity 		:= lrVelocity,
					Acceleration 	:= lrAcceleration,
					Deceleration 	:= lrDeceleration,
					Jerk 			:= lrJerk,
					BufferMode 		:= eBufferMode);

IF fbMcMoveAbsolute.Error THEN
	bError := TRUE;
	bMoveActive := FALSE;
	iErrorID := fbMcMoveAbsolute.ErrorID;
	fbMcMoveAbsolute( Axis := stAxisRef, Execute := FALSE);
	fbAlarmMoveAbsolute.ipArguments.Clear().AddUDInt(iErrorID);
	fbAlarmMoveAbsolute.Raise(0);

ELSIF fbMcMoveAbsolute.Done THEN
	eAxisState := AXIS_MOVE_ABSOLUTE_DONE;
END_IF
END_METHOD

METHOD PROTECTED MS_MoveAbsoluteDone
VAR_INPUT
END_VAR
fbMcMoveAbsolute( Axis := stAxisRef, Execute := FALSE);

IF NOT bMoveAbsolute AND NOT fbMcMoveAbsolute.Busy THEN
	eAxisState := AXIS_IDLE;
END_IF
END_METHOD

METHOD PROTECTED MS_MoveAdditive
VAR_INPUT
END_VAR
fbMcMoveAdditive(	Axis			:= stAxisRef,
					Execute 		:= TRUE,
					Distance 		:= lrRelativeDistance,
					Velocity		:= lrVelocity,
					Acceleration	:= lrAcceleration,
					Deceleration	:= lrDeceleration,
					Jerk			:= lrJerk,
					BufferMode 		:= eBufferMode);

IF fbMcMoveAdditive.Error THEN
	bError := TRUE;
	bMoveActive := FALSE;
	iErrorID := fbMcMoveAdditive.ErrorID;
	fbMcMoveAdditive( Axis := stAxisRef, Execute := FALSE);
	fbAlarmMoveAdditive.ipArguments.Clear().AddUDInt(iErrorID);
	fbAlarmMoveAdditive.Raise(0);
		
ELSIF fbMcMoveAdditive.Done THEN
	eAxisState := AXIS_MOVE_ADDITIVE_DONE;
END_IF
END_METHOD

METHOD PROTECTED MS_MoveAdditiveDone
VAR_INPUT
END_VAR
fbMcMoveAdditive( Axis := stAxisRef, Execute := FALSE);

IF NOT bMoveAdditive AND NOT fbMcMoveAdditive.Busy THEN
	eAxisState := AXIS_IDLE;
END_IF
END_METHOD

METHOD PROTECTED MS_MoveJog
VAR_INPUT
END_VAR
VAR
	bJogForward: BOOL;
	bJogBackward: BOOL;
END_VAR
IF eJogDirection = AXIS_JOG_DIR_POSITIVE THEN
	bJogForward := TRUE;
	bJogBackward:= FALSE;
	
ELSIF eJogDirection = AXIS_JOG_DIR_NEGATIVE THEN
	bJogForward := FALSE;
	bJogBackward:= TRUE;
		
END_IF

fbMcJog( 	Axis 			:= stAxisRef,
			JogForward		:= bJogForward,
			JogBackwards	:= bJogBackward,
			Mode 			:= eJogMode,
			Position 		:= lrJogPosition,
			Velocity 		:= lrJogVelocity,
			Acceleration 	:= lrJogAcceleration,
			Deceleration 	:= lrJogDeceleration,
			Jerk 			:= lrJogJerk);

IF fbMcJog.Error THEN
	bError := TRUE;
	bMoveActive := FALSE;
	iErrorID := fbMcJog.ErrorID;
	fbMcJog( Axis := stAxisRef, JogForward := FALSE, JogBackwards := FALSE);
	fbAlarmMoveJog.ipArguments.Clear().AddUDInt(iErrorID);
	fbAlarmMoveJog.Raise(0);
	
ELSIF fbMcJog.Mode >= MC_JOGMODE_INCHING AND fbMcJog.Done THEN
	eAxisState := AXIS_MOVE_JOG_DONE;
		
ELSIF fbMcJog.Mode < MC_JOGMODE_INCHING AND NOT bJogActive THEN
	eAxisState := AXIS_MOVE_JOG_DONE;
		
END_IF
END_METHOD

METHOD PROTECTED MS_MoveJogDone
VAR_INPUT
END_VAR
fbMcJog( Axis := stAxisRef, JogForward := FALSE, JogBackwards := FALSE);

IF NOT bJog AND NOT fbMcJog.Busy THEN
	eAxisState := AXIS_IDLE;
END_IF
END_METHOD

METHOD PROTECTED MS_MoveRelative
VAR_INPUT
END_VAR
fbMcMoveRelative(	Axis 			:= stAxisRef,
					Execute 		:= TRUE,
					Distance 		:= lrRelativeDistance,
					Velocity 		:= lrVelocity,
					Acceleration 	:= lrAcceleration,
					Deceleration 	:= lrDeceleration,
					Jerk 			:= lrJerk,
					BufferMode 		:= eBufferMode);
				
IF fbMcMoveRelative.Error THEN
	bError := TRUE;
	iErrorID := fbMcMoveRelative.ErrorID;
	fbMcMoveRelative( Axis := stAxisRef, Execute := FALSE);
	fbAlarmMoveRelative.ipArguments.Clear().AddUDInt(iErrorID);
	fbAlarmMoveRelative.Raise(0);
	
ELSIF fbMcMoveRelative.Done THEN
	eAxisState := AXIS_MOVE_RELATIVE_DONE;
END_IF
END_METHOD

METHOD PROTECTED MS_MoveRelativeDone
VAR_INPUT
END_VAR
fbMcMoveRelative( Axis := stAxisRef, Execute := FALSE);

IF NOT bMoveRelative AND NOT fbMcMoveRelative.Busy THEN
	bInPostion := TRUE;
	bInVelocity := FALSE;
	bMoveActive := FALSE;
	bStopped := FALSE;
	bHalted := FALSE;
	bJogDone := FALSE;
	eAxisState := AXIS_IDLE;
END_IF
END_METHOD

METHOD PROTECTED MS_MoveVelocity
VAR_INPUT
END_VAR
fbMcMoveVelocity(	Axis 			:= stAxisRef,
					Execute 		:= TRUE,
					Velocity 		:= lrVelocity,
					Acceleration 	:= lrAcceleration,
					Deceleration 	:= lrDeceleration,
					Jerk 			:= lrJerk,
					Direction 		:= eDirection,
					BufferMode 		:= eBufferMode);

IF fbMcMoveVelocity.Error THEN
	bError := TRUE;
	iErrorID := fbMcMoveVelocity.ErrorID;
	fbMcMoveVelocity( Axis := stAxisRef, Execute := FALSE);
	fbAlarmMoveVelocity.ipArguments.Clear().AddUDInt(iErrorID);
	fbAlarmMoveVelocity.Raise(0);
	
ELSIF fbMcMoveVelocity.InVelocity THEN
	eAxisState := AXIS_MOVE_VELOCITY_DONE;
END_IF
END_METHOD

METHOD PROTECTED MS_MoveVelocityDone
VAR_INPUT
END_VAR
fbMcMoveVelocity( Axis := stAxisRef, Execute := FALSE);

IF NOT bMoveVelocity AND NOT fbMcMoveVelocity.Busy THEN
	eAxisState := AXIS_IDLE;
END_IF
END_METHOD

METHOD PROTECTED MS_ReadyInitialized
VAR_INPUT
END_VAR
eAxisState := AXIS_IDLE;
END_METHOD

METHOD PROTECTED MS_Reset
VAR_INPUT
END_VAR
(* Reset MC_Halt *)
fbMcHalt( Axis := stAxisRef, Execute := FALSE);

(* Reset MC_Stop *)
fbMcStop( Axis := stAxisRef, Execute := FALSE);

(* Reset MC_MoveVelocity *)
fbMcMoveVelocity( Axis := stAxisRef, Execute := FALSE);

(* Reset MC_MoveAbsolute *)
fbMcMoveAbsolute( Axis := stAxisRef, Execute := FALSE);

(* Reset MC_MoveAdditive *)
fbMcMoveAdditive( Axis := stAxisRef, Execute := FALSE);

(* Reset MC_MoveRelative *)
fbMcMoveRelative( Axis := stAxisRef, Execute := FALSE);

(* Reset MC_Jog *)
fbMcJog( Axis := stAxisRef, JogForward := FALSE ,JogBackwards := FALSE);

(* Reset MC_GearIn *)
;

(* Reset MC_GearOut *)
;

(* Reset internal commands *)
bAbort			:= FALSE;
bHalt 			:= FALSE;
bHome			:= FALSE;
bJog			:= FALSE;
bMoveAbsolute	:= FALSE;
bMoveAdditive	:= FALSE;
bMoveRelative	:= FALSE;
bMoveVelocity	:= FALSE;
bStop			:= FALSE;

fbMcReset( Axis := stAxisRef, Execute := TRUE);

IF fbMcReset.Error THEN
	bError := TRUE;
	iErrorID := fbMcReset.ErrorID;
	fbMcReset( Axis := stAxisRef, Execute := FALSE);
	fbAlarmInitReset.ipArguments.Clear().AddUDInt(iErrorID);
	fbAlarmInitReset.Raise(0);
	
ELSIF fbMcReset.Done THEN
	fbMcReset(Axis := stAxisRef, Execute := FALSE);
	
	(* Confirming and resetting alarms *)
	fbAlarmHalt.Confirm(nTimeStamp := 0);
	fbAlarmInitReset.Confirm(nTimeStamp := 0);
	fbAlarmInitPowerOn.Confirm(nTimeStamp := 0);
	fbAlarmMoveAbsolute.Confirm(nTimeStamp := 0);
	fbAlarmMoveAdditive.Confirm(nTimeStamp := 0);
	fbAlarmMoveJog.Confirm(nTimeStamp := 0);
	fbAlarmMoveRelative.Confirm(nTimeStamp := 0);
	fbAlarmMoveVelocity.Confirm(nTimeStamp := 0);
	fbAlarmStop.Confirm(nTimeStamp := 0);
	fbAlarmHome.Confirm(nTimeStamp := 0);
	fbAlarmHaltCA.Confirm(nTimeStamp := 0);
	fbAlarmMoveAbsoluteCA.Confirm(nTimeStamp := 0);
	fbAlarmMoveRelativeCA.Confirm(nTimeStamp := 0);
	fbAlarmCoupling.Confirm(nTimeStamp := 0);
	fbAlarmDecoupling.Confirm(nTimeStamp := 0);

	fbAlarmHalt.Clear(nTimeStamp := 0, bResetConfirmation := bResetConfirmation); 
	fbAlarmInitReset.Clear(nTimeStamp := 0, bResetConfirmation := bResetConfirmation); 
	fbAlarmInitPowerOn.Clear(nTimeStamp := 0, bResetConfirmation := bResetConfirmation); 
	fbAlarmMoveAbsolute.Clear(nTimeStamp := 0, bResetConfirmation := bResetConfirmation); 
	fbAlarmMoveAdditive.Clear(nTimeStamp := 0, bResetConfirmation := bResetConfirmation); 
	fbAlarmMoveJog.Clear(nTimeStamp := 0, bResetConfirmation := bResetConfirmation); 
	fbAlarmMoveRelative.Clear(nTimeStamp := 0, bResetConfirmation := bResetConfirmation); 
	fbAlarmMoveVelocity.Clear( nTimeStamp := 0, bResetConfirmation := bResetConfirmation); 
	fbAlarmStop.Clear(nTimeStamp := 0, bResetConfirmation := bResetConfirmation); 
	fbAlarmHome.Clear(nTimeStamp := 0, bResetConfirmation := bResetConfirmation); 
	fbAlarmHaltCA.Clear(nTimeStamp := 0, bResetConfirmation := bResetConfirmation); 
	fbAlarmMoveAbsoluteCA.Clear(nTimeStamp := 0, bResetConfirmation := bResetConfirmation); 
	fbAlarmMoveRelativeCA.Clear(nTimeStamp := 0, bResetConfirmation := bResetConfirmation); 
	fbAlarmCoupling.Clear(nTimeStamp := 0, bResetConfirmation := bResetConfirmation); 
	fbAlarmDecoupling.Clear(nTimeStamp := 0, bResetConfirmation := bResetConfirmation); 

	IF NOT fbMcHalt.Busy AND NOT fbMcStop.Busy AND NOT fbMcMoveVelocity.Busy AND
		NOT fbMcMoveAbsolute.Busy AND NOT fbMcMoveAdditive.Busy AND NOT fbMcMoveRelative.Busy AND NOT fbMcReset.Busy THEN
		eAxisState := AXIS_RESET_DONE;
	END_IF
END_IF
END_METHOD

METHOD PROTECTED MS_ResetDone
VAR_INPUT
END_VAR
IF NOT bReset THEN
	IF eAxisStateBeforeReset >= E_AxisState.AXIS_IDLE THEN
		eAxisState := AXIS_IDLE;
	ELSE
		eAxisState := AXIS_UNINITIALIZED;	
	END_IF
END_IF
END_METHOD

METHOD PROTECTED MS_Stop
VAR_INPUT
END_VAR
(* Reset MC_MoveVelocity *)
fbMcMoveVelocity( Axis := stAxisRef, Execute := FALSE);

(* Reset MC_MoveAbsolute *)					
fbMcMoveAbsolute( Axis := stAxisRef, Execute := FALSE);

(* Reset MC_MoveAdditive *)					
fbMcMoveAdditive( Axis := stAxisRef ,Execute := FALSE);

(* Reset MC_MoveRelative *)					
fbMcMoveRelative( Axis := stAxisRef, Execute := FALSE);

(* Reset MC_Jog *)
fbMcJog( Axis := stAxisRef, JogForward := FALSE, JogBackwards := FALSE);

fbMcStop(	Execute 		:= TRUE,
			Axis 			:= stAxisRef,
			Deceleration	:= lrStopDeceleration,
			Jerk 			:= lrStopJerk);

IF fbMcStop.Error THEN
	bError := TRUE;
	iErrorID := fbMcStop.ErrorID;
	fbMcStop( Axis := stAxisRef, Execute := FALSE);
	fbAlarmStop.ipArguments.Clear().AddUDInt(iErrorID);
	fbAlarmStop.Raise(0);
	
ELSIF fbMcStop.Done THEN
	eAxisState := AXIS_STOP_DONE;
END_IF
END_METHOD

METHOD PROTECTED MS_StopDone
VAR_INPUT
END_VAR
fbMcStop( Axis := stAxisRef, Execute := FALSE);

IF NOT bStop THEN
	eAxisState := AXIS_IDLE;	
END_IF
END_METHOD

METHOD PROTECTED MS_Uninitalized
VAR_INPUT
END_VAR
(* Reset all commands *)
bAbort				:= FALSE;
bHalt 				:= FALSE;
bHome				:= FALSE;
bJog				:= FALSE;
bMoveAbsolute		:= FALSE;
bMoveAdditive		:= FALSE;
bMoveRelative		:= FALSE;
bMoveVelocity		:= FALSE;
bReset				:= FALSE;
bStop				:= FALSE;

(* Reset status flags *)
bError				:= FALSE;
bInPostion			:= FALSE;
bInVelocity			:= FALSE;
bIsHomed			:= FALSE;
bMoveActive			:= FALSE;
bPowerOn			:= FALSE;
bStopped			:= FALSE;
bJogDone			:= FALSE;
bLocked				:= FALSE;
lrActualPosition 	:= 0.0;
lrActualVelocity 	:= 0.0;
iErrorID			:= 0;

IF bInit THEN
	eAxisState := AXIS_INITIALIZING;
	eAxisStateInit := AXIS_INIT_RESET;	
END_IF
END_METHOD

METHOD MS_Unlock
VAR_INPUT
END_VAR
fbMcStop( Axis := stAxisRef, Execute := FALSE);

IF NOT fbMcStop.Busy THEN
	eAxisState := AXIS_UNLOCK_DONE;
END_IF
END_METHOD

METHOD MS_UnlockDone
VAR_INPUT
END_VAR
IF NOT bUnlock THEN
	eAxisState := AXIS_IDLE;
END_IF
END_METHOD

PROPERTY Name : STRING
GET
Name := sName;
END_GET
SET
sName := Name;
END_SET
END_PROPERTY

PROPERTY Options : Tc2_MC2.ST_MoveOptions
GET
Options := stOptions;
END_GET
SET
stOptions := Options;
END_SET
END_PROPERTY

PROPERTY Override : LREAL
GET
Override := lrOverride;
END_GET
SET
IF Override >= 0.0 AND Override <= 200.0 THEN
	lrOverride := Override;
	fbMcPower( Axis := stAxisRef, Override := lrOverride);
END_IF
END_SET
END_PROPERTY

PROPERTY PowerOn : REFERENCE TO BOOL
GET
PowerOn REF= bPowerOn;
END_GET
END_PROPERTY

PROPERTY SetpointPosition : LREAL
GET
SetpointPosition := stAxisRef.NcToPlc.SetPos;
END_GET
END_PROPERTY

PROPERTY SetpointVelocity : LREAL
GET
SetpointVelocity := stAxisRef.NcToPlc.SetVelo;
END_GET
END_PROPERTY

PROPERTY State : REFERENCE TO E_AxisState
GET
State REF= eAxisState;
END_GET
END_PROPERTY

METHOD PROTECTED StateMachine
VAR_INPUT
END_VAR

VAR

END_VAR
CASE eAxisState OF
	AXIS_UNINITIALIZED:
		MS_Uninitalized();
		
	AXIS_INITIALIZING:
		MS_Initializing();
		
	AXIS_READY_INITIALIZED:
		MS_ReadyInitialized();
		
	AXIS_IDLE:
		MS_Idle();
	
	AXIS_HOME:
		MS_Home();
		
	E_AxisState.AXIS_HOME_DONE:
		MS_HomeDone();
		
	AXIS_MOVE_VELOCITY:
		MS_MoveVelocity();
	
	AXIS_MOVE_VELOCITY_DONE:
		MS_MoveVelocityDone();
	
	AXIS_MOVE_ABSOLUTE:
		MS_MoveAbsolute();
	
	AXIS_MOVE_ABSOLUTE_DONE:
		MS_MoveAbsoluteDone();
	
	AXIS_MOVE_ADDITIVE:
		MS_MoveAdditive();
	
	AXIS_MOVE_ADDITIVE_DONE:
		MS_MoveAdditiveDone();
		
	AXIS_MOVE_RELATIVE:
		MS_MoveRelative();
		
	AXIS_MOVE_RELATIVE_DONE:
		MS_MoveRelativeDone();
	
	AXIS_MOVE_JOG:
		MS_MoveJog();
	
	AXIS_MOVE_JOG_DONE:
		MS_MoveJogDone();
	
	AXIS_STOP:
		MS_Stop();
	
	AXIS_STOP_DONE:
		MS_StopDone();
		
	AXIS_HALT:
		MS_Halt();
	
	AXIS_HALT_DONE:
		MS_HaltDone();	
	
	AXIS_RESET:
		MS_Reset();
	
	AXIS_RESET_DONE:
		MS_ResetDone();
		
	AXIS_ABORTING:
		MS_Aborting();
		
	AXIS_COUPLE:
		MS_Couple();
		
	AXIS_COUPLE_DONE:
		MS_CoupleDone();
		
	AXIS_DECOUPLE:
		MS_Decouple();
		
	AXIS_DECOUPLE_DONE:
		MS_DecoupleDone();
		
	AXIS_UNLOCK:
		MS_Unlock();
	
	AXIS_UNLOCK_DONE:
		MS_UnlockDone();
		
	AXIS_EXTENSION:
		MS_Extension();
		
END_CASE
END_METHOD

PROPERTY StatePlcOpen : REFERENCE TO E_AxisStatePlcOpen
GET
StatePlcOpen REF= eStatePlcOpen;
END_GET
END_PROPERTY

PROPERTY StopDeceleration : LREAL
GET
StopDeceleration := lrStopDeceleration;
END_GET
SET
lrStopDeceleration := StopDeceleration;
END_SET
END_PROPERTY

PROPERTY StopJerk : LREAL
GET
StopJerk := lrStopJerk;
END_GET
SET
lrStopJerk := StopJerk;
END_SET
END_PROPERTY

PROPERTY Stopped : REFERENCE TO BOOL
GET
Stopped REF= bStopped;
END_GET
END_PROPERTY

PROPERTY Unit : STRING
GET
Unit := sUnit;
END_GET
SET
sUnit := Unit;
END_SET
END_PROPERTY

PROPERTY Velocity : LREAL
GET
Velocity := lrVelocity;
END_GET
SET
lrVelocity := Velocity;
END_SET
END_PROPERTY

END_FUNCTION_BLOCK

// ---- POUs/Axis/FB_AxisServoCA.TcPOU
(* 
:Description: This function block is used represent basic axis controled by standard PLCopen motion function blocks with collision avoidance feature.
*)
FUNCTION_BLOCK FB_AxisServoCA EXTENDS FB_AxisServo IMPLEMENTS I_UniversalAxisCA
VAR
	(*Commands *)
	bHaltCA				: BOOL;	(*  *)
	bMoveAbsoluteCA		: BOOL;	(*  *)
	bMoveRelativeCA		: BOOL;	(*  *)
	bHaltedCA			: BOOL;
	
	(* Parameters *)
	lrGap				: MC_LREAL;
	eDirectionCa		: Tc3_Mc3Definitions.MC_DIRECTION; (* Axis movement direction for collision avoidance *)
	stMoveAbsCaOptions	: ST_MoveAbsoluteCAOptions;
		
	(* Function blocks *)
	fbMcHaltCA			: MC_HaltCA;			(* Halt with colision avoidance *)
	fbMcMoveAbsoluteCA	: MC_MoveAbsoluteCA;	(* Move absolute with colision avoidance *)
	fbMcMoveRelativeCA	: MC_MoveRelativeCA;	(* Move relative with colision avoidance *)
	
	eAxisStateCA		: E_AxisStateCA;		(*  *)
	tonDelay			: TON;				(* Delay which allows to see any page changes during tests *)

END_VAR

IF bFirstCycle THEN
	stMoveAbsCaOptions.GapControlMode := MC_GAP_CONTROL_MODE.mcGapControlModeStandard;
END_IF

SUPER^();

tonDelay();

PROPERTY DirectionCA : Tc3_Mc3Definitions.MC_DIRECTION
GET
DirectionCA := eDirectionCa;
END_GET
SET
eDirectionCa := DirectionCA;
END_SET
END_PROPERTY

PROPERTY Gap : MC_LREAL
GET
Gap := lrGap;
END_GET
SET
lrGap := Gap;
END_SET
END_PROPERTY

PROPERTY HaltedCA : REFERENCE TO BOOL
GET
HaltedCA REF= bHaltedCA;
END_GET
END_PROPERTY

METHOD MR_HaltCA : BOOL
VAR_INPUT
END_VAR
IF eAxisState >= AXIS_IDLE AND eAxisStateCA <> AXIS_CA_HALT_DONE THEN
	bHaltedCA := FALSE;
	
	IF NOT bHaltLog THEN 
		fbMachineLogger.MR_AddLogs(CONCAT(sName,' : halt (CA) requested'));
		bHaltLog := TRUE;
	END_IF
	
	bHaltCA := TRUE;
	MR_HaltCA := FALSE;
	eAxisState := AXIS_EXTENSION;
	eAxisStateCA := AXIS_CA_HALT;
	
ELSIF eAxisState = AXIS_EXTENSION AND eAxisStateCA = AXIS_CA_HALT_DONE THEN
	bInPostion 	:= FALSE;
	bInVelocity := FALSE;
	bMoveActive := FALSE;
	bStopped 	:= FALSE;
	bJogDone 	:= FALSE;
	bHaltedCA	:= TRUE;
	
	bHaltCA		:= FALSE;
	MR_HaltCA 	:= TRUE;
	bHaltLog 	:= FALSE;
	fbMachineLogger.MR_AddLogs(CONCAT(sName,' : halt (CA) done'));
	
END_IF
END_METHOD

METHOD MR_MoveAbsoluteCA : BOOL
VAR_INPUT
	lrAbsolutePosition : LREAL;
END_VAR
VAR
	bFirstCycle		   : BOOL := TRUE;
END_VAR
VAR_INST
	lrAbsolutePositionTemp : LREAL;
END_VAR
IF bFirstCycle THEN
	bFirstCycle := FALSE;
	
	IF THIS^.lrAbsolutePosition = lrAbsolutePosition THEN
		lrAbsolutePositionTemp := lrAbsolutePosition - 0.001;
		
	ELSE
		lrAbsolutePositionTemp := lrAbsolutePosition;
		
	END_IF
END_IF


IF eAxisState = AXIS_IDLE AND THIS^.lrAbsolutePosition <> lrAbsolutePositionTemp THEN
	THIS^.lrAbsolutePosition := lrAbsolutePosition;
	bInPostion 	:= FALSE;
	bInVelocity := FALSE;
	bMoveActive := TRUE;
	bStopped 	:= FALSE;
	bHalted 	:= FALSE;
	bJogDone 	:= FALSE;
	bHaltedCA 	:= FALSE;
	
	bMoveAbsoluteCA := TRUE;
	MR_MoveAbsoluteCA := FALSE;
	eAxisState := AXIS_EXTENSION;
	eAxisStateCA := AXIS_CA_MOVE_ABSOLUTE;
	fbMachineLogger.MR_AddLogs(CONCAT(sName,' : move absoulte (CA) requested'));		
	
ELSIF eAxisState = AXIS_EXTENSION AND eAxisStateCA = AXIS_CA_MOVE_ABSOLUTE_DONE THEN
	bInPostion 		:= TRUE;
	bInVelocity		:= FALSE;
	bMoveActive 	:= FALSE;
	bStopped 		:= FALSE;
	bHalted			:= FALSE;
	bJogDone 		:= FALSE;
	bHaltedCA 		:= TRUE;
	
	bMoveAbsoluteCA := FALSE;
	MR_MoveAbsoluteCA := TRUE;
	fbMachineLogger.MR_AddLogs(CONCAT(sName,' : move absoulte (CA) done'));		
	
END_IF
END_METHOD

METHOD MR_MoveRelativeCA : BOOL
VAR_INPUT
	lrRelativeDistance : LREAL;
END_VAR
IF eAxisState = AXIS_IDLE AND lrRelativeDistance <> 0.0 THEN
	bInPostion 	:= FALSE;
	
	THIS^.lrRelativeDistance := lrRelativeDistance;
	bInVelocity := FALSE;
	bMoveActive := TRUE;
	bStopped 	:= FALSE;
	bHalted 	:= FALSE;
	bJogDone 	:= FALSE;
	bHaltedCA 	:= FALSE;
	
	bMoveRelativeCA := TRUE;
	MR_MoveRelativeCA := FALSE;
	eAxisState := AXIS_EXTENSION;
	eAxisStateCA := AXIS_CA_MOVE_RELATIVE;
	fbMachineLogger.MR_AddLogs(CONCAT(sName,' : move relative (CA) requested'));			
	
ELSIF eAxisState = AXIS_EXTENSION AND eAxisStateCA = AXIS_CA_MOVE_RELATIVE_DONE THEN
	bInVelocity 	:= FALSE;
	bMoveActive 	:= FALSE;
	bStopped 		:= FALSE;
	bHalted 		:= FALSE;
	bJogDone 		:= FALSE;
	bHaltedCA 		:= TRUE;
	
	bMoveRelativeCA := FALSE;
	MR_MoveRelativeCA := TRUE;
	bInPostion 		:= TRUE;
	fbMachineLogger.MR_AddLogs(CONCAT(sName,' : move relative (CA) done'));		
	
END_IF
END_METHOD

METHOD PROTECTED MS_Aborting
VAR_INPUT
END_VAR
(* Reset MC_MoveAbsoluteCA *)
fbMcMoveAbsoluteCA( Axis := stAxisRef, Execute := FALSE);

(* Reset MC_MoveRelativeCA *)
fbMcMoveRelativeCA( Axis := stAxisRef, Execute := FALSE);

(* Reset MC_HaltCA *)
fbMcHaltCA( Axis := stAxisRef, Execute := FALSE);

(* Run parent deinitializing procedure *)
SUPER^.MS_Aborting();
END_METHOD

METHOD MS_AxisCAIdle : BOOL
VAR_INPUT
END_VAR
;
END_METHOD

METHOD MS_Extension : BOOL
VAR_INPUT
END_VAR
CASE eAxisStateCA OF
	E_AxisStateCA.AXIS_CA_IDLE:
		MS_AxisCAIdle();
		
	E_AxisStateCA.AXIS_CA_MOVE_ABSOLUTE:
		MS_MoveAbsoluteCA();
		
	E_AxisStateCA.AXIS_CA_MOVE_ABSOLUTE_DONE:
		MS_MoveAbsoluteCADone();
		
	E_AxisStateCA.AXIS_CA_MOVE_RELATIVE:
		MS_MoveRelativeCA();
		
	E_AxisStateCA.AXIS_CA_MOVE_RELATIVE_DONE:
		MS_MoveRelativeCADone();
		
	E_AxisStateCA.AXIS_CA_HALT:
		MS_HaltCA();
		
	E_AxisStateCA.AXIS_CA_HALT_DONE:
		MS_HaltDoneCA();
	
END_CASE
END_METHOD

METHOD PROTECTED MS_HaltCA
VAR_INPUT
END_VAR
fbMcHaltCA( Axis			:= stAxisRef,
			Execute			:= TRUE,
			Deceleration	:= lrDeceleration,
			Gap				:= lrGap);
	
IF fbMcHaltCA.Error THEN
	bError := TRUE;
	iErrorID := fbMcHaltCA.ErrorId;
	fbMcHaltCA( Axis := stAxisRef, Execute := FALSE);	
	fbAlarmHaltCA.ipArguments.Clear().AddUDInt(iErrorID);	
	fbAlarmHaltCA.Raise(0);

ELSIF fbMcHaltCA.Done THEN
	fbMcMoveAbsoluteCA( Axis := stAxisRef, Execute := FALSE);
	eAxisStateCA := AXIS_CA_HALT_DONE;
	bHalted 	:= TRUE;
	
END_IF
END_METHOD

METHOD PROTECTED MS_HaltDoneCA
VAR_INPUT
END_VAR
(* Reset MC_HaltCA *)
fbMcHaltCA( Axis := stAxisRef, Execute := FALSE);	

IF NOT bHaltCA AND NOT fbMcHaltCA.Busy THEN
	tonDelay(IN := TRUE, PT:= T#200MS);
	
	IF tonDelay.Q THEN
		tonDelay(IN := FALSE);
		eAxisState := AXIS_IDLE;
		eAxisStateCA := AXIS_CA_IDLE;
		
	END_IF
END_IF
END_METHOD

METHOD MS_MoveAbsoluteCA : BOOL
VAR_INPUT
END_VAR
CASE eAxesGroupMethodState OF
	AXES_GROUP_METHOD_EXECUTE:
		fbMcMoveAbsoluteCA(	Axis			:= stAxisRef,
							Execute			:= TRUE,
							Velocity		:= lrVelocity,
							Position		:= lrAbsolutePosition,
							Acceleration	:= lrAcceleration,
							Deceleration	:= lrDeceleration,
							Jerk			:= lrJerk,
							Gap				:= lrGap,
							Direction		:= eDirectionCa,
							Options			:= stMoveAbsCaOptions);

		IF NOT fbMcMoveAbsoluteCA.Busy THEN
			eAxesGroupMethodState := AXES_GROUP_METHOD_DONE; 
			
		END_IF
	
	AXES_GROUP_METHOD_DONE:
		IF fbMcMoveAbsoluteCA.Error THEN
			bError := TRUE;
			iErrorID := fbMcMoveAbsoluteCA.ErrorId;
			fbMcMoveAbsoluteCA( Axis := stAxisRef, Execute := FALSE);
			fbAlarmMoveAbsoluteCA.ipArguments.Clear().AddUDInt(iErrorID);
			fbAlarmMoveAbsoluteCA.Raise(0);
				
		ELSE //fbMcMoveAbsoluteCA.Done THEN
			eAxisStateCA := AXIS_CA_MOVE_ABSOLUTE_DONE;
			
		END_IF
END_CASE
END_METHOD

METHOD MS_MoveAbsoluteCADone : BOOL
VAR_INPUT
END_VAR
(* Reset MC_MoveAbsoluteCA *)
fbMcMoveAbsoluteCA( Axis := stAxisRef, Execute := FALSE);

IF bInPostion THEN
	eAxisState := AXIS_IDLE;
 	eAxesGroupMethodState := AXES_GROUP_METHOD_EXECUTE;
	eAxisStateCA := AXIS_CA_IDLE;
	
END_IF
END_METHOD

METHOD PROTECTED MS_MoveRelativeCA
VAR_INPUT
END_VAR
CASE eAxesGroupMethodState OF
	AXES_GROUP_METHOD_EXECUTE:
		fbMcMoveRelativeCA(	Axis			:= stAxisRef,
							Execute			:= TRUE,
							Distance		:= lrRelativeDistance,
							Velocity		:= lrVelocity,
							Acceleration	:= lrAcceleration,
							Deceleration	:= lrDeceleration,
							Jerk			:= lrJerk,
							Gap 			:= lrGap);

		IF NOT fbMcMoveRelativeCA.Busy THEN
			eAxesGroupMethodState := AXES_GROUP_METHOD_DONE; 
			
		END_IF
							
							
	AXES_GROUP_METHOD_DONE:						
		IF fbMcMoveRelativeCA.Error THEN
			bError := TRUE;
			iErrorID := fbMcMoveRelativeCA.ErrorId;
			fbMcMoveRelativeCA( Axis := stAxisRef, Execute := FALSE);
			fbAlarmMoveRelativeCA.ipArguments.Clear().AddUDInt(iErrorID);
			fbAlarmMoveRelativeCA.Raise(0);
			
		ELSE //fbMcMoveRelativeCA.Done THEN
			eAxisStateCA := AXIS_CA_MOVE_RELATIVE_DONE;
				
		END_IF
END_CASE
END_METHOD

METHOD PROTECTED MS_MoveRelativeCADone
VAR_INPUT
END_VAR
(* Reset MC_MoveRelativeCA *)
fbMcMoveRelativeCA( Axis := stAxisRef, Execute := FALSE);

IF bInPostion THEN
	eAxisState := AXIS_IDLE;
	eAxisStateCA := AXIS_CA_IDLE;
 	eAxesGroupMethodState := AXES_GROUP_METHOD_EXECUTE;

END_IF
END_METHOD

(* 
Copyrights	: Sonion Industrialization - Control Systems Desing Department
Author		: Adrian Bogdzia - based on MEMS universal libraries
Date		: 11/2021
Description : This function block is used represent basic axis
*)
METHOD PROTECTED MS_Reset
VAR_INPUT
END_VAR
(* Reset MC_MoveAbsoluteCA *)
fbMcMoveAbsoluteCA( Axis := stAxisRef, Execute := FALSE);

(* Reset MC_MoveRelativeCA *)
fbMcMoveRelativeCA( Axis := stAxisRef, Execute := FALSE);

(* Reset MC_HaltCA *)
fbMcHaltCA( Axis := stAxisRef, Execute := FALSE);

(* Run parent reset procedure *)
SUPER^.MS_Reset();
END_METHOD

METHOD PROTECTED MS_Stop
VAR_INPUT
END_VAR
(* Reset MC_MoveAbsoluteCA *)
fbMcMoveAbsoluteCA( Axis := stAxisRef, Execute := FALSE);

(* Reset MC_MoveRelativeCA *)
fbMcMoveRelativeCA( Axis := stAxisRef, Execute := FALSE);

(* Run parent stop procedure *)
SUPER^.MS_Stop();
END_METHOD

PROPERTY StateCA : REFERENCE TO E_AxisStateCA
GET
StateCA REF= eAxisStateCA;
END_GET
END_PROPERTY

END_FUNCTION_BLOCK
